//! <summary>Reports the concrete instance size in bytes, excluding separately allocated storage.</summary>
{attribute 'monitoring' := 'call'}
PROPERTY SelfSize : ULINT
GET
SelfSize := XSIZEOF(THIS^);
END_GET
END_PROPERTY

END_FUNCTION_BLOCK

// ---- Tests/Files/FileByteOperationsTest.TcPOU
(*
SPDX-FileCopyrightText: © 2026 Oleksandr Tiutyk <trofimich@gmail.com>
SPDX-License-Identifier: MIT
License: https://opensource.org/license/mit
*)

(*!
<summary>Exercises queued binary I/O and standalone collision, load, rename and delete operations.</summary>
<description>
Uses one exclusive directory and bounded persistent buffers. Checks short read, EOF, tell and guarded results
before and after cancellation. Independent directory probes must preserve the sentinel file. Rename and delete
are followed by readback and a failed load. Direct operations are drained before the base attempts removal.
Use from one task and keep the case alive until cleanup finishes. Do not copy this test.
</description>
*)

{attribute 'no_assign'}
{attribute 'no_explicit_call' := 'do not call this function block directly'}
FUNCTION_BLOCK FileByteOperationsTest EXTENDS FileContentScenarioTest
VAR_STAT
	//! <summary>Class name shared by instances of this concrete function block.</summary>
	{attribute 'hide'}
	_ClassName : STRING := __POUNAME();
END_VAR
VAR CONSTANT
	//! <summary>Truncates the file and permits binary writes and reads through the same handle.</summary>
	_UpdateBinaryMode : DWORD := Tc2_System.Global_Variables.FOPEN_MODEWRITE
		OR Tc2_System.Global_Variables.FOPEN_MODEPLUS
		OR Tc2_System.Global_Variables.FOPEN_MODEBINARY;
	//! <summary>Marks bytes beyond the written range so partial and empty reads can detect stray writes.</summary>
	_UnusedByte : BYTE := BYTE#16#A5;
END_VAR
VAR
	_Phase : FILE_OPERATIONS_TEST_PHASE;
	_ReusedTask : TOF_Tasks.ITask;
	_Write : TOF_FileSystem.WriteBytesToFile(name := "Write four bytes");
	_TellAfterWrite : TOF_FileSystem.GetPositionInFile(name := "Tell after write");
	_Seek : TOF_FileSystem.SetPositionInFile(name := "Rewind binary file");
	_Read : TOF_FileSystem.ReadBytesFromFile(name := "Short binary read");
	_TellAfterRead : TOF_FileSystem.GetPositionInFile(name := "Tell after read");
	_ReadEof : TOF_FileSystem.ReadBytesFromFile(name := "Read past EOF");
	_CheckEof : TOF_FileSystem.CheckEndOfFile(name := "Check EOF");

	_CheckDirectory : TOF_FileSystem.CheckDirectoryExists(name := "Check file as directory");
	_CreateIfAbsent : TOF_FileSystem.CreateDirectoryIfNotExists(name := "Create on file collision");
	_RemoveIfPresent : TOF_FileSystem.RemoveEmptyDirectoryIfExists(name := "Remove on file collision");
	_CreateExisting : TOF_FileSystem.CreateDirectory(name := "Create existing directory");
	_Load : TOF_FileSystem.LoadFile(name := "Load binary file");
	_Rename : TOF_FileSystem.RenameFile(name := "Rename binary file");
	_Delete : TOF_FileSystem.DeleteFile(name := "Delete binary file");

	_ResultTasks : ARRAY [0..5] OF TOF_Tasks.ITask :=
		[_Write, _TellAfterWrite, _Read, _TellAfterRead, _ReadEof, _CheckEof];
	_CollisionTasks : ARRAY [0..3] OF TOF_Tasks.ITask :=
		[_CheckDirectory, _CreateIfAbsent, _RemoveIfPresent, _CreateExisting];

	_Data : ARRAY [0..3] OF BYTE := [BYTE#16#41, BYTE#16#42, BYTE#16#43, BYTE#16#44];
	_ReadBuffer : ARRAY [0..7] OF BYTE;
	_LoadBuffer : ARRAY [0..7] OF BYTE;
	_EofBuffer : BYTE;
END_VAR

(*!
<summary>Rearms the direct and queued tasks and restores the initial binary buffers.</summary>
*)
METHOD PROTECTED ResetScenario : BOOL
VAR
	i : DINT;
END_VAR
_Phase := FILE_OPERATIONS_TEST_PHASE.START_WRITE;
_ReusedTask := 0;
_EofBuffer := _UnusedByte;

FOR i := LOWER_BOUND(_ReadBuffer, 1) TO UPPER_BOUND(_ReadBuffer, 1) DO
	_ReadBuffer[i] := _UnusedByte;
END_FOR

FOR i := LOWER_BOUND(_ResultTasks, 1) TO UPPER_BOUND(_ResultTasks, 1) DO
	IF NOT _ResultTasks[i].Reset() THEN
		RETURN;
	END_IF
END_FOR

FOR i := LOWER_BOUND(_CollisionTasks, 1) TO UPPER_BOUND(_CollisionTasks, 1) DO
	IF NOT _CollisionTasks[i].Reset() THEN
		RETURN;
	END_IF
END_FOR

ResetScenario := _Seek.Reset() AND_THEN _Load.Reset() AND_THEN _Rename.Reset() AND_THEN _Delete.Reset();
END_METHOD

(*!
<summary>Drains direct and pre-submission cancellation tasks before owned directory removal.</summary>
<description>The base invokes this after the manager stops. Every eligible task is advanced on each call.</description>
*)
METHOD PROTECTED DrainScenario : BOOL
VAR
	i : DINT;
END_VAR
DrainScenario := TRUE;

FOR i := LOWER_BOUND(_CollisionTasks, 1) TO UPPER_BOUND(_CollisionTasks, 1) DO
	DrainScenario := drainTask(task := _CollisionTasks[i]) AND DrainScenario;
END_FOR

IF _ReusedTask <> 0 THEN
	DrainScenario := drainTask(task := _ReusedTask) AND DrainScenario;
END_IF

DrainScenario := drainTask(task := _Load) AND DrainScenario;
DrainScenario := drainTask(task := _Rename) AND DrainScenario;
DrainScenario := drainTask(task := _Delete) AND DrainScenario;
END_METHOD

(*!
<summary>Requests cooperative cancellation and advances an active task one cycle.</summary>
<param name="task">Live task that is no longer controlled by the file manager.</param>
*)
METHOD PRIVATE drainTask : BOOL
VAR_INPUT
	task : TOF_Tasks.ITask;
END_VAR
IF task.State.Running THEN
	task.Cancel();
	task.Execute();
END_IF

drainTask := NOT task.State.Running;
END_METHOD

(*!
<summary>Advances the native byte, collision and path-operation phases.</summary>
<description>Returns TRUE after the final missing-file check. The base handles reporting after cleanup.</description>
*)
METHOD PROTECTED AdvanceScenario : BOOL
VAR
	i : DINT;
END_VAR
CASE _Phase OF
	FILE_OPERATIONS_TEST_PHASE.START_WRITE:
		startByteQueue();

	FILE_OPERATIONS_TEST_PHASE.WAIT_FOR_WRITE:
		_Manager.Execute();

		IF _Write.State.Running THEN
			CheckScenario(
				condition := _Write.ActuallyWrittenBytes = TOF_Core.UnsignedInt32.ZERO,
				message := "RUNNING write must hide its byte count"
			);
		END_IF

		IF _Read.State.Running THEN
			CheckScenario(
				condition := _Read.ActuallyReadBytes = TOF_Core.UnsignedInt32.ZERO AND_THEN NOT _Read.IsEndOfFile,
				message := "RUNNING read must hide its byte count and EOF"
			);
		END_IF

		IF _TellAfterWrite.State.Running THEN
			CheckScenario(
				condition := _TellAfterWrite.Position = TOF_Core.SignedInt32.ZERO,
				message := "RUNNING tell must hide its file position"
			);
		END_IF

		IF _Manager.State.Stopped AND_THEN _ScenarioFailure = "" THEN
			IF checkWorkDone(task := _Manager) THEN
				checkByteResults();
			END_IF

			_Phase := FILE_OPERATIONS_TEST_PHASE.CHECK_COLLISIONS;
		END_IF

	FILE_OPERATIONS_TEST_PHASE.CHECK_COLLISIONS:
		startCollisions();

	FILE_OPERATIONS_TEST_PHASE.WAIT_FOR_COLLISIONS:
		IF checkCollisions() THEN
			_Phase := FILE_OPERATIONS_TEST_PHASE.START_LOAD;
		END_IF

	FILE_OPERATIONS_TEST_PHASE.START_LOAD:
		_Load.TargetBuffer := ADR(_LoadBuffer);
		_Load.TargetBufferSize := SIZEOF(_LoadBuffer);
		_Load.Timeout := _NativeTimeout;
		startLoad(filePath := _Directory.FirstFilePath);
		_Phase := FILE_OPERATIONS_TEST_PHASE.WAIT_FOR_LOAD;

	FILE_OPERATIONS_TEST_PHASE.WAIT_FOR_LOAD:
		_Load.Execute();

		IF _Load.State.Running THEN
			CheckScenario(
				condition := _Load.LoadedBytesCount = TOF_Core.UnsignedInt32.ZERO,
				message := "RUNNING load must hide its byte count"
			);
		ELSIF _Load.State.Stopped AND_THEN checkWorkDone(task := _Load) THEN
			checkLoadedBytes(context := "File after collision attempts");
			_Phase := FILE_OPERATIONS_TEST_PHASE.START_RENAME;
		END_IF

	FILE_OPERATIONS_TEST_PHASE.START_RENAME:
		_Directory.ExpectSecondFile();
		_Rename.OldFilePath := _Directory.FirstFilePath;
		_Rename.NewFilePath := _Directory.SecondFilePath;
		_Rename.PathType := Tc2_System.E_OpenPath.PATH_GENERIC;
		_Rename.Timeout := _NativeTimeout;
		CheckScenario(condition := _Rename.Start(), message := "Rename refused Start");
		_Phase := FILE_OPERATIONS_TEST_PHASE.WAIT_FOR_RENAME;

	FILE_OPERATIONS_TEST_PHASE.WAIT_FOR_RENAME:
		_Rename.Execute();

		IF _Rename.State.Stopped AND_THEN checkWorkDone(task := _Rename) THEN
			_Directory.ConfirmFirstFileAbsent();
			_Phase := FILE_OPERATIONS_TEST_PHASE.LOAD_RENAMED_FILE;
		END_IF

	FILE_OPERATIONS_TEST_PHASE.LOAD_RENAMED_FILE:
		startLoad(filePath := _Directory.SecondFilePath);
		_Phase := FILE_OPERATIONS_TEST_PHASE.WAIT_FOR_RENAMED_LOAD;

	FILE_OPERATIONS_TEST_PHASE.WAIT_FOR_RENAMED_LOAD:
		_Load.Execute();

		IF _Load.State.Stopped AND_THEN checkWorkDone(task := _Load) THEN
			checkLoadedBytes(context := "Renamed file");
			_Phase := FILE_OPERATIONS_TEST_PHASE.START_DELETE;
		END_IF

	FILE_OPERATIONS_TEST_PHASE.START_DELETE:
		_Delete.FilePath := _Directory.SecondFilePath;
		_Delete.PathType := Tc2_System.E_OpenPath.PATH_GENERIC;
		_Delete.Timeout := _NativeTimeout;
		CheckScenario(condition := _Delete.Start(), message := "Delete refused Start");
		_Phase := FILE_OPERATIONS_TEST_PHASE.WAIT_FOR_DELETE;

	FILE_OPERATIONS_TEST_PHASE.WAIT_FOR_DELETE:
		_Delete.Execute();

		IF _Delete.State.Stopped AND_THEN checkWorkDone(task := _Delete) THEN
			_Directory.ConfirmSecondFileAbsent();
			_Phase := FILE_OPERATIONS_TEST_PHASE.LOAD_DELETED_FILE;
		END_IF

	FILE_OPERATIONS_TEST_PHASE.LOAD_DELETED_FILE:
		startLoad(filePath := _Directory.SecondFilePath);
		_Phase := FILE_OPERATIONS_TEST_PHASE.WAIT_FOR_MISSING_LOAD;

	FILE_OPERATIONS_TEST_PHASE.WAIT_FOR_MISSING_LOAD:
		_Load.Execute();

		IF _Load.State.Stopped THEN
			CheckScenario(
				condition := _Load.FinalStopReason.Failure
					AND_THEN _Load.LoadedBytesCount = TOF_Core.UnsignedInt32.ZERO,
				message := "Load of a deleted file must fail and expose zero bytes"
			);

			FOR i := LOWER_BOUND(_LoadBuffer, 1) TO UPPER_BOUND(_LoadBuffer, 1) DO
				IF _LoadBuffer[i] <> _UnusedByte THEN
					CheckScenario(
						condition := FALSE,
						message := TOF_Core.WideStrings.ConcatFit255("Missing-file load altered buffer byte ", TO_WSTRING(i))
					);
					RETURN;
				END_IF
			END_FOR

			AdvanceScenario := TRUE;
		END_IF
END_CASE
END_METHOD

(*!
<summary>Configures and starts the binary write, seek, read and position queue.</summary>
<description>The directory is owned and all borrowed queue tasks are READY.</description>
*)
METHOD PRIVATE startByteQueue
_Directory.ExpectFirstFile();
ConfigureFile(filePath := _Directory.FirstFilePath, modeFlags := _UpdateBinaryMode);
_Write.SourceBuffer := ADR(_Data);
_Write.BytesCountToWrite := SIZEOF(_Data);
_Write.Timeout := _NativeTimeout;
_TellAfterWrite.Timeout := _NativeTimeout;
_Seek.Position := TOF_Core.SignedInt32.ZERO;
_Seek.Origin := Tc2_System.E_SeekOrigin.SEEK_SET;
_Seek.Timeout := _NativeTimeout;
_Read.TargetBuffer := ADR(_ReadBuffer);
_Read.BytesCountToRead := SIZEOF(_ReadBuffer);
_Read.Timeout := _NativeTimeout;
_TellAfterRead.Timeout := _NativeTimeout;
_ReadEof.TargetBuffer := ADR(_EofBuffer);
_ReadEof.BytesCountToRead := SIZEOF(_EofBuffer);
_ReadEof.Timeout := _NativeTimeout;
_CheckEof.Timeout := _NativeTimeout;

_Manager.Enqueue(fileHandleTask := _Write);
_Manager.Enqueue(fileHandleTask := _TellAfterWrite);
_Manager.Enqueue(fileHandleTask := _Seek);
_Manager.Enqueue(fileHandleTask := _Read);
_Manager.Enqueue(fileHandleTask := _TellAfterRead);
_Manager.Enqueue(fileHandleTask := _ReadEof);
_Manager.Enqueue(fileHandleTask := _CheckEof);

CheckScenario(
	condition := _Write.ActuallyWrittenBytes = TOF_Core.UnsignedInt32.ZERO,
	message := "READY write must expose zero bytes"
);
CheckScenario(
	condition := _Read.ActuallyReadBytes = TOF_Core.UnsignedInt32.ZERO AND_THEN NOT _Read.IsEndOfFile,
	message := "READY read must expose zero bytes and FALSE EOF"
);
CheckScenario(condition := NOT _CheckEof.IsEndOfFile, message := "READY EOF query must expose FALSE");

IF _ScenarioFailure = "" THEN
	CheckScenario(condition := _Manager.Start(), message := "Binary write/read queue refused Start");
	_Phase := FILE_OPERATIONS_TEST_PHASE.WAIT_FOR_WRITE;
END_IF
END_METHOD

(*!
<summary>Verifies the readback and neutral results after pre-submission cancellation.</summary>
<description>Call after the manager completes the full queue and releases the resource.</description>
*)
METHOD PRIVATE checkByteResults
VAR
	i : DINT;
	task : TOF_Tasks.ITask;
END_VAR
CheckScenario(
	condition := _Write.ActuallyWrittenBytes = 4,
	message := "Full write must report four bytes"
);
CheckScenario(condition := _Read.ActuallyReadBytes = 4, message := "Short read must report the actual four bytes");
CheckScenario(condition := _TellAfterWrite.Position = 4, message := "Tell after write must report position four");
CheckScenario(condition := _TellAfterRead.Position = 4, message := "Tell after short read must report position four");
CheckScenario(
	condition := _ReadEof.ActuallyReadBytes = TOF_Core.UnsignedInt32.ZERO AND_THEN _ReadEof.IsEndOfFile,
	message := "Read past the data must return zero bytes and TRUE EOF"
);
CheckScenario(condition := _CheckEof.IsEndOfFile, message := "EOF query after empty read must report TRUE");
CheckScenario(condition := _EofBuffer = _UnusedByte, message := "Empty read must preserve its destination");

FOR i := LOWER_BOUND(_Data, 1) TO UPPER_BOUND(_Data, 1) DO
	CheckScenario(
		condition := _ReadBuffer[i] = _Data[i],
		message := TOF_Core.WideStrings.ConcatFit255("Binary readback differs at byte ", TO_WSTRING(i))
	);
END_FOR

FOR i := UPPER_BOUND(_Data, 1) + 1 TO UPPER_BOUND(_ReadBuffer, 1) DO
	CheckScenario(
		condition := _ReadBuffer[i] = _UnusedByte,
		message := TOF_Core.WideStrings.ConcatFit255("Short read altered buffer tail at byte ", TO_WSTRING(i))
	);
END_FOR

IF _ScenarioFailure <> "" THEN
	RETURN;
END_IF

FOR i := LOWER_BOUND(_ResultTasks, 1) TO UPPER_BOUND(_ResultTasks, 1) DO
	task := _ResultTasks[i];
	_ReusedTask := task;

	IF NOT task.Reset() OR_ELSE NOT task.Start() OR_ELSE NOT task.Cancel() THEN
		_ScenarioFailure := TOF_Core.WideStrings.ConcatFit255(task.Name, " refused Reset, Start or Cancel during reuse");
		RETURN;
	END_IF

	task.Execute();

	IF NOT task.State.Stopped OR_ELSE NOT task.FinalStopReason.ExternalCancel THEN
		_ScenarioFailure := TOF_Core.WideStrings.ConcatFit255(
			task.Name, " did not stop with pre-submission cancellation"
		);
		RETURN;
	END_IF

	_ReusedTask := 0;
END_FOR

CheckScenario(
	condition := _Write.ActuallyWrittenBytes = TOF_Core.UnsignedInt32.ZERO,
	message := "Cancelled write exposed its previous byte count"
);
CheckScenario(
	condition := _Read.ActuallyReadBytes = TOF_Core.UnsignedInt32.ZERO,
	message := "Cancelled read exposed its previous byte count"
);
CheckScenario(
	condition := _TellAfterWrite.Position = TOF_Core.SignedInt32.ZERO
		AND_THEN _TellAfterRead.Position = TOF_Core.SignedInt32.ZERO,
	message := "Cancelled tell exposed its previous file position"
);
CheckScenario(condition := NOT _ReadEof.IsEndOfFile, message := "Cancelled read exposed its previous TRUE EOF");
CheckScenario(
	condition := NOT _CheckEof.IsEndOfFile,
	message := "Cancelled EOF query exposed its previous TRUE EOF"
);
END_METHOD

(*!
<summary>Starts directory probes against the existing sentinel file and its parent.</summary>
<description>Only the original fixture owns the directory. All four probes borrow paths only.</description>
*)
METHOD PRIVATE startCollisions
VAR
	i : DINT;
END_VAR
_CheckDirectory.DirectoryPath := _Directory.FirstFilePath;
_CreateIfAbsent.DirectoryPath := _Directory.FirstFilePath;
_RemoveIfPresent.DirectoryPath := _Directory.FirstFilePath;
_CreateExisting.DirectoryPath := _Directory.DirectoryPath;
_CheckDirectory.PathType := Tc2_System.E_OpenPath.PATH_GENERIC;
_CreateIfAbsent.PathType := Tc2_System.E_OpenPath.PATH_GENERIC;
_RemoveIfPresent.PathType := Tc2_System.E_OpenPath.PATH_GENERIC;
_CreateExisting.PathType := Tc2_System.E_OpenPath.PATH_GENERIC;
_CheckDirectory.Timeout := _NativeTimeout;
_CreateIfAbsent.Timeout := _NativeTimeout;
_RemoveIfPresent.Timeout := _NativeTimeout;
_CreateExisting.Timeout := _NativeTimeout;

FOR i := LOWER_BOUND(_CollisionTasks, 1) TO UPPER_BOUND(_CollisionTasks, 1) DO
	IF NOT _CollisionTasks[i].Start() THEN
		_ScenarioFailure := TOF_Core.WideStrings.ConcatFit255(_CollisionTasks[i].Name, " refused Start");
		RETURN;
	END_IF
END_FOR

_Phase := FILE_OPERATIONS_TEST_PHASE.WAIT_FOR_COLLISIONS;
END_METHOD

(*!
<summary>Advances outstanding collision probes and verifies their stopped results.</summary>
<description>Returns TRUE after all four operations stop with the expected outcomes.</description>
*)
METHOD PRIVATE checkCollisions : BOOL
VAR
	i : DINT;
	allStopped : BOOL := TRUE;
END_VAR
FOR i := LOWER_BOUND(_CollisionTasks, 1) TO UPPER_BOUND(_CollisionTasks, 1) DO
	IF _CollisionTasks[i].State.Running THEN
		_CollisionTasks[i].Execute();
	END_IF

	allStopped := allStopped AND _CollisionTasks[i].State.Stopped;
END_FOR

IF NOT allStopped THEN
	RETURN;
END_IF

IF NOT checkWorkDone(task := _CheckDirectory) THEN
	RETURN;
END_IF

CheckScenario(condition := NOT _CheckDirectory.DirectoryExists, message := "A file was reported as a directory");
CheckScenario(
	condition := _CreateIfAbsent.FinalStopReason.Failure,
	message := "Conditional directory creation did not reject the file collision"
);
CheckScenario(
	condition := _RemoveIfPresent.FinalStopReason.Failure,
	message := "Conditional directory removal did not reject the file collision"
);
CheckScenario(
	condition := _CreateExisting.FinalStopReason.Failure,
	message := "Ordinary directory creation did not reject the existing directory"
);
checkCollisions := _ScenarioFailure = "";
END_METHOD

(*!
<summary>Resets the load task, refills its target and starts loading the specified file.</summary>
<param name="filePath">Owned fixture path to load, including the deliberate missing-file check.</param>
*)
METHOD PRIVATE startLoad
VAR_INPUT
	filePath : Tc2_System.T_MaxString;
END_VAR
VAR
	i : DINT;
END_VAR
IF NOT _Load.Reset() THEN
	_ScenarioFailure := "File load refused Reset";
	RETURN;
END_IF

IF _Load.LoadedBytesCount <> TOF_Core.UnsignedInt32.ZERO THEN
	_ScenarioFailure := "READY file load exposed its previous byte count";
	RETURN;
END_IF

FOR i := LOWER_BOUND(_LoadBuffer, 1) TO UPPER_BOUND(_LoadBuffer, 1) DO
	_LoadBuffer[i] := _UnusedByte;
END_FOR

_Load.FilePath := filePath;
CheckScenario(condition := _Load.Start(), message := "File load refused Start");
END_METHOD

(*!
<summary>Checks the full sentinel and the untouched tail of a successful load.</summary>
<param name="context">Operation that preceded this readback.</param>
*)
METHOD PRIVATE checkLoadedBytes
VAR_INPUT
	context : WSTRING(80);
END_VAR
VAR
	i : DINT;
END_VAR
CheckScenario(
	condition := _Load.LoadedBytesCount = 4,
	message := TOF_Core.WideStrings.ConcatFit255(context, ": expected four loaded bytes")
);

FOR i := LOWER_BOUND(_Data, 1) TO UPPER_BOUND(_Data, 1) DO
	CheckScenario(
		condition := _LoadBuffer[i] = _Data[i],
		message := TOF_Core.WideStrings.ConcatFit255(context, ": sentinel differs at byte ", TO_WSTRING(i))
	);
END_FOR

FOR i := UPPER_BOUND(_Data, 1) + 1 TO UPPER_BOUND(_LoadBuffer, 1) DO
	CheckScenario(
		condition := _LoadBuffer[i] = _UnusedByte,
		message := TOF_Core.WideStrings.ConcatFit255(context, ": load altered buffer tail at byte ", TO_WSTRING(i))
	);
END_FOR
END_METHOD

(*!
<summary>Reports the task name and copied stop diagnostic when a native operation fails.</summary>
<param name="task">Stopped task whose success is required to continue.</param>
*)
METHOD PRIVATE checkWorkDone : BOOL
VAR_INPUT
	task : TOF_Tasks.ITask;
END_VAR
checkWorkDone := task.FinalStopReason.WorkDone;

IF NOT checkWorkDone AND_THEN _ScenarioFailure = "" THEN
	_ScenarioFailure := TOF_Core.WideStrings.ConcatFit255(task.Name, " did not finish with WorkDone: ");
	TOF_Core.WideStrings.AppendFit(targetString := _ScenarioFailure, sourceString := task.FinalStopReason.Message);
END_IF
END_METHOD

//! <summary>Borrows the concrete type name; callers must not modify the referenced storage.</summary>
{attribute 'monitoring' := 'call'}
PROPERTY ClassName : REFERENCE TO STRING
GET
ClassName REF= _ClassName;
END_GET
END_PROPERTY

//! <summary>Borrows the compiler-initialized namespace; callers must not modify it.</summary>
{attribute 'monitoring' := 'call'}
PROPERTY NamespaceName : REFERENCE TO STRING
GET
NamespaceName REF= CurrentNamespace.Name;
END_GET
END_PROPERTY

//! <summary>Reports the concrete instance size in bytes, excluding separately allocated storage.</summary>
{attribute 'monitoring' := 'call'}
PROPERTY SelfSize : ULINT
GET
SelfSize := XSIZEOF(THIS^);
END_GET
END_PROPERTY

END_FUNCTION_BLOCK

// ---- Tests/Files/FileBinaryBufferMatrixTest.TcPOU
(*
SPDX-FileCopyrightText: © 2026 Oleksandr Tiutyk <trofimich@gmail.com>
SPDX-License-Identifier: MIT
License: https://opensource.org/license/mit
*)

(*!
<summary>Checks six invalid binary buffer configurations on an acquired file resource.</summary>
<description>
Uses an owned file and opens a fresh update handle for each row. Verifies the configured property diagnostic,
neutral public results, intact caller data and resource release. No sampled cycle may report native busy;
native tracing is needed to rule out a submission that completed between observations.
Use from one task and do not copy this test.
</description>
*)

{attribute 'no_assign'}
{attribute 'no_explicit_call' := 'do not call this function block directly'}
FUNCTION_BLOCK FileBinaryBufferMatrixTest EXTENDS FileContentScenarioTest
VAR_STAT
	//! <summary>Class name shared by instances of this concrete function block.</summary>
	{attribute 'hide'}
	_ClassName : STRING := __POUNAME();
END_VAR
VAR CONSTANT
	//! <summary>First row using WriteBytesToFile. The preceding three rows use ReadBytesFromFile.</summary>
	_FirstWriteRow : DINT := 3;
	//! <summary>Total number of null and zero sized buffer configurations under test.</summary>
	_RowCount : DINT := 6;
	//! <summary>Identifies unexpected changes to caller-owned storage in each invalid row.</summary>
	_BufferSentinel : BYTE := BYTE#16#A5;
	//! <summary>Creates a new, empty binary file before the validation rows.</summary>
	_CreateBinaryMode : DWORD := Tc2_System.Global_Variables.FOPEN_MODEWRITE
		OR Tc2_System.Global_Variables.FOPEN_MODEBINARY;
	//! <summary>Reopens the existing file for binary reads and writes without truncating it.</summary>
	_OpenBinaryMode : DWORD := Tc2_System.Global_Variables.FOPEN_MODEREAD
		OR Tc2_System.Global_Variables.FOPEN_MODEPLUS
		OR Tc2_System.Global_Variables.FOPEN_MODEBINARY;
END_VAR
VAR
	_Phase : FILE_BUFFER_TEST_PHASE;
	_Read : TOF_FileSystem.ReadBytesFromFile(name := "Invalid read buffer");
	_Write : TOF_FileSystem.WriteBytesToFile(name := "Invalid write buffer");
	_Operation : TOF_Tasks.ITask;
	_ExpectedProperty : STRING(32);
	_Row : DINT;
	_Buffer : BYTE;
END_VAR

(*!
<summary>Rearms the binary operations and restarts the matrix from its first row.</summary>
*)
METHOD PROTECTED ResetScenario : BOOL
_Phase := FILE_BUFFER_TEST_PHASE.CREATE_FILE;
_Operation := 0;
_Row := 0;
ResetScenario := _Read.Reset() AND_THEN _Write.Reset();
END_METHOD

(*!
<summary>Creates the fixture file and advances one invalid buffer row at a time.</summary>
<description>Queues the invalid child only after acquisition is observed. Returns TRUE after the sixth row.</description>
*)
METHOD PROTECTED AdvanceScenario : BOOL
CASE _Phase OF
	FILE_BUFFER_TEST_PHASE.CREATE_FILE:
		_Directory.ExpectFirstFile();
		ConfigureFile(filePath := _Directory.FirstFilePath, modeFlags := _CreateBinaryMode);
		CheckScenario(condition := _Manager.Start(), message := "Creating the matrix file refused Start");
		_Phase := FILE_BUFFER_TEST_PHASE.WAIT_FOR_FILE;

	FILE_BUFFER_TEST_PHASE.WAIT_FOR_FILE:
		_Manager.Execute();

		IF _Manager.State.Stopped THEN
			IF NOT _Manager.FinalStopReason.WorkDone OR_ELSE _Manager.ResourceManager.ResourceAcquired THEN
				_ScenarioFailure := "Creating the matrix file did not finish and release the resource: ";
				TOF_Core.WideStrings.AppendFit(
					targetString := _ScenarioFailure,
					sourceString := _Manager.FinalStopReason.Message
				);
				RETURN;
			END_IF

			_Phase := FILE_BUFFER_TEST_PHASE.START_INVALID_OPERATION;
		END_IF

	FILE_BUFFER_TEST_PHASE.START_INVALID_OPERATION:
		startRow();

	FILE_BUFFER_TEST_PHASE.WAIT_FOR_INVALID_OPERATION:
		_Manager.Execute();

		IF _Manager.State.Stopped THEN
			IF NOT checkRow() THEN
				RETURN;
			END_IF

			_Row := _Row + 1;
			AdvanceScenario := _Row = _RowCount;
			_Phase := FILE_BUFFER_TEST_PHASE.START_INVALID_OPERATION;
		ELSIF _Read.FileOperationInProgress OR_ELSE _Write.FileOperationInProgress THEN
			failRow(reason := "an invalid buffer exposed a pending native request");
		ELSIF _Manager.ResourceManager.ResourceAcquired
			AND_THEN _Manager.RunningSubstate.Processing
			AND_THEN _Manager.PendingTaskCount = 0
			AND_THEN _Operation.State.Ready
		THEN
			IF _Row < _FirstWriteRow THEN
				_Manager.Enqueue(fileHandleTask := _Read);
			ELSE
				_Manager.Enqueue(fileHandleTask := _Write);
			END_IF

			_Manager.StopWhenNoPendingTasks := TRUE;
		END_IF
END_CASE
END_METHOD

(*!
<summary>Configures one null or zero buffer combination and starts acquiring its file.</summary>
<description>Called with no active file operation, after creating the file or checking the previous row.</description>
*)
METHOD PRIVATE startRow
IF NOT _Manager.Reset() OR_ELSE NOT _Read.Reset() OR_ELSE NOT _Write.Reset() THEN
	_ScenarioFailure := TOF_Core.WideStrings.ConcatFit255(
		"Buffer row ", TO_WSTRING(_Row + 1), ": the manager or a binary operation refused Reset"
	);
	RETURN;
END_IF

ConfigureFile(filePath := _Directory.FirstFilePath, modeFlags := _OpenBinaryMode);
_Manager.StopWhenNoPendingTasks := FALSE;
_Buffer := _BufferSentinel;
_Read.Timeout := _NativeTimeout;
_Write.Timeout := _NativeTimeout;
_Read.TargetBuffer := TOF_Core.Memory.NULL_ADDRESS;
_Read.BytesCountToRead := TOF_Core.UnsignedInt32.ZERO;
_Write.SourceBuffer := TOF_Core.Memory.NULL_ADDRESS;
_Write.BytesCountToWrite := TOF_Core.UnsignedInt32.ZERO;

CASE _Row OF
	0:
		_Read.BytesCountToRead := 1;
		_ExpectedProperty := 'TargetBuffer';
	1:
		_Read.TargetBuffer := ADR(_Buffer);
		_ExpectedProperty := 'BytesCountToRead';
	2:
		_ExpectedProperty := 'TargetBuffer';
	3:
		_Write.BytesCountToWrite := 1;
		_ExpectedProperty := 'SourceBuffer';
	4:
		_Write.SourceBuffer := ADR(_Buffer);
		_ExpectedProperty := 'BytesCountToWrite';
	5:
		_ExpectedProperty := 'SourceBuffer';
END_CASE

IF _Row < _FirstWriteRow THEN
	_Operation := _Read;
ELSE
	_Operation := _Write;
END_IF

IF NOT _Manager.Start() THEN
	failRow(reason := "the update file manager refused Start");
	RETURN;
END_IF

_Phase := FILE_BUFFER_TEST_PHASE.WAIT_FOR_INVALID_OPERATION;
END_METHOD

(*!
<summary>Verifies the actual child failure, release and data after the manager stops.</summary>
<description>Returns TRUE for a failed child with its expected property diagnostic and no retained resource.</description>
*)
METHOD PRIVATE checkRow : BOOL
VAR
	diagnostic : STRING(255);
END_VAR
IF NOT _Operation.State.Stopped OR_ELSE NOT _Operation.FinalStopReason.Failure THEN
	failRow(reason := "the invalid child did not reach STOPPED with Failure");
	TOF_Core.WideStrings.AppendFit(targetString := _ScenarioFailure, sourceString := " | Manager: ");
	TOF_Core.WideStrings.AppendFit(targetString := _ScenarioFailure, sourceString := _Manager.FinalStopReason.Message);
	RETURN;
END_IF

IF NOT _Manager.FinalStopReason.Failure OR_ELSE _Manager.ResourceManager.ResourceAcquired THEN
	failRow(reason := "the manager did not report Failure with the resource released");
	RETURN;
END_IF

IF _Read.FileOperationInProgress OR_ELSE _Write.FileOperationInProgress THEN
	failRow(reason := "native I/O was still pending after the manager stopped");
	RETURN;
END_IF

IF _Buffer <> _BufferSentinel
	OR_ELSE _Read.ActuallyReadBytes <> TOF_Core.UnsignedInt32.ZERO
	OR_ELSE _Write.ActuallyWrittenBytes <> TOF_Core.UnsignedInt32.ZERO
	OR_ELSE _Read.IsEndOfFile
THEN
	failRow(reason := "the invalid operation altered caller data or exposed a non-neutral result");
	RETURN;
END_IF

diagnostic := TO_STRING(_Operation.FinalStopReason.Message);

IF NOT TOF_Core.Strings.Contains(stringToSearchIn := diagnostic, stringToFind := _ExpectedProperty) THEN
	failRow(reason := "the child diagnostic did not name the expected public property");
	TOF_Core.WideStrings.AppendFit(targetString := _ScenarioFailure, sourceString := " | Actual: ");
	TOF_Core.WideStrings.AppendFit(targetString := _ScenarioFailure, sourceString := _Operation.FinalStopReason.Message);
	RETURN;
END_IF

checkRow := TRUE;
END_METHOD

(*!
<summary>Copies the matrix row, expected property and its first failure for deferred reporting.</summary>
<param name="reason">Condition that failed before cooperative cleanup.</param>
*)
METHOD PRIVATE failRow
VAR_INPUT
	reason : WSTRING(255);
END_VAR
_ScenarioFailure := TOF_Core.WideStrings.ConcatFit255(
	"Buffer row ", TO_WSTRING(_Row + 1), " (", TO_WSTRING(_ExpectedProperty), "): ", reason
);
END_METHOD

//! <summary>Borrows the concrete type name; callers must not modify the referenced storage.</summary>
{attribute 'monitoring' := 'call'}
PROPERTY ClassName : REFERENCE TO STRING
GET
ClassName REF= _ClassName;
END_GET
END_PROPERTY

//! <summary>Borrows the compiler-initialized namespace; callers must not modify it.</summary>
{attribute 'monitoring' := 'call'}
PROPERTY NamespaceName : REFERENCE TO STRING
GET
NamespaceName REF= CurrentNamespace.Name;
END_GET
END_PROPERTY

//! <summary>Reports the concrete instance size in bytes, excluding separately allocated storage.</summary>
{attribute 'monitoring' := 'call'}
PROPERTY SelfSize : ULINT
GET
SelfSize := XSIZEOF(THIS^);
END_GET
END_PROPERTY

END_FUNCTION_BLOCK

// ---- Tests/Files/FileCallerExceptionCleanupTest.TcPOU
(*
SPDX-FileCopyrightText: © 2026 Oleksandr Tiutyk <trofimich@gmail.com>
SPDX-License-Identifier: MIT
License: https://opensource.org/license/mit
*)

(*!
<summary>Verifies cooperative release after an exception in the file manager's caller.</summary>
<description>
Raises a known StandardException only while the file resource is acquired. The caller catches and checks its
identity, then requests cancellation on a later cycle and drives the manager to STOPPED. The base removes the
owned artifacts before publishing a result. Native resource state does not certify physical close.
Use from one task and do not copy this test.
</description>
*)

{attribute 'no_assign'}
{attribute 'no_explicit_call' := 'do not call this function block directly'}
FUNCTION_BLOCK FileCallerExceptionCleanupTest EXTENDS FileContentScenarioTest
VAR_STAT
	//! <summary>Class name shared by instances of this concrete function block.</summary>
	{attribute 'hide'}
	_ClassName : STRING := __POUNAME();
END_VAR
VAR CONSTANT
	//! <summary>Payload used to distinguish the deliberate caller fault from unrelated exceptions.</summary>
	_CallerMessage : WSTRING(255) := "Synthetic exception in the file-scenario caller";
	//! <summary>Creates an empty owned file for observing acquisition and cancellation.</summary>
	_CreateBinaryMode : DWORD := Tc2_System.Global_Variables.FOPEN_MODEWRITE
		OR Tc2_System.Global_Variables.FOPEN_MODEBINARY;
END_VAR
VAR
	_Phase : FILE_CALLER_CLEANUP_TEST_PHASE;
END_VAR

(*!
<summary>Restores the opening phase after the base rearms the manager.</summary>
*)
METHOD PROTECTED ResetScenario : BOOL
_Phase := FILE_CALLER_CLEANUP_TEST_PHASE.OPEN_FILE;
ResetScenario := TRUE;
END_METHOD

(*!
<summary>Opens a file, catches the caller fault and continues cancellation until release.</summary>
<description>Returns TRUE after observing STOPPED and checking the final reason and resource state.</description>
*)
METHOD PROTECTED AdvanceScenario : BOOL
CASE _Phase OF
	FILE_CALLER_CLEANUP_TEST_PHASE.OPEN_FILE:
		_Directory.ExpectFirstFile();
		ConfigureFile(filePath := _Directory.FirstFilePath, modeFlags := _CreateBinaryMode);
		_Manager.StopWhenNoPendingTasks := FALSE;
		CheckScenario(condition := _Manager.Start(), message := "Caller-exception manager refused Start");
		_Phase := FILE_CALLER_CLEANUP_TEST_PHASE.INJECT_CALLER_EXCEPTION;

	FILE_CALLER_CLEANUP_TEST_PHASE.INJECT_CALLER_EXCEPTION:
		_Manager.Execute();

		IF _Manager.State.Running
			AND_THEN _Manager.ResourceManager.ResourceAcquired
			AND_THEN _Manager.RunningSubstate.Processing
		THEN
			CheckScenario(
				condition := catchCallerException(),
				message := "Expected caller exception was not caught intact"
			);
			_Phase := FILE_CALLER_CLEANUP_TEST_PHASE.DRAIN_MANAGER;
		ELSIF _Manager.State.Stopped THEN
			_ScenarioFailure := "Caller fault requires an acquired file resource: ";
			TOF_Core.WideStrings.AppendFit(
				targetString := _ScenarioFailure,
				sourceString := _Manager.FinalStopReason.Message
			);
		END_IF

	FILE_CALLER_CLEANUP_TEST_PHASE.DRAIN_MANAGER:
		IF _Manager.RunningSubstate.Processing AND_THEN NOT _Manager.Cancel() THEN
			_ScenarioFailure := "The acquired manager refused caller cancellation";
			RETURN;
		END_IF

		_Manager.Execute();

		IF _Manager.State.Stopped THEN
			IF NOT _Manager.FinalStopReason.ExternalCancel THEN
				_ScenarioFailure := "Caller recovery did not stop with ExternalCancel: ";
				TOF_Core.WideStrings.AppendFit(
					targetString := _ScenarioFailure,
					sourceString := _Manager.FinalStopReason.Message
				);
				RETURN;
			END_IF

			CheckScenario(
				condition := NOT _Manager.ResourceManager.ResourceAcquired,
				message := "Caller recovery left the file resource acquired"
			);
			AdvanceScenario := TRUE;
		END_IF
END_CASE
END_METHOD

(*!
<summary>Injects and recognises the deliberate exception outside the manager's Execute call.</summary>
<description>Returns TRUE only for the expected standard payload. No exception reference survives this call.</description>
*)
METHOD PRIVATE catchCallerException : BOOL
VAR
	exceptionCode : __SYSTEM.ExceptionCode;
	caughtException : TOF_Core.IException;
	standardException : TOF_Core.IStandardException;
	message : TOF_Core.ERROR_MESSAGE;
END_VAR
message := _CallerMessage;

__TRY
	TOF_Core.Exceptions.ThrowStandard(
		sourceNamespaceName := NamespaceName,
		sourceClassName := ClassName,
		sourcePOUName := __POUNAME(),
		sourcePosition := __POSITION(),
		message := message
	);
__CATCH(exceptionCode)
	caughtException := TOF_Core.ExceptionManager.GetLastException(
		exceptionCode := exceptionCode,
		catchPointNamespaceName := NamespaceName,
		catchPointPOUName := __POUNAME(),
		catchPointPosition := __POSITION()
	);
	catchCallerException := __QUERYINTERFACE(caughtException, standardException)
		AND_THEN standardException.SourceMessage = _CallerMessage;
__ENDTRY
END_METHOD

//! <summary>Borrows the concrete type name; callers must not modify the referenced storage.</summary>
{attribute 'monitoring' := 'call'}
PROPERTY ClassName : REFERENCE TO STRING
GET
ClassName REF= _ClassName;
END_GET
END_PROPERTY

//! <summary>Borrows the compiler-initialized namespace; callers must not modify it.</summary>
{attribute 'monitoring' := 'call'}
PROPERTY NamespaceName : REFERENCE TO STRING
GET
NamespaceName REF= CurrentNamespace.Name;
END_GET
END_PROPERTY

//! <summary>Reports the concrete instance size in bytes, excluding separately allocated storage.</summary>
{attribute 'monitoring' := 'call'}
PROPERTY SelfSize : ULINT
GET
SelfSize := XSIZEOF(THIS^);
END_GET
END_PROPERTY

END_FUNCTION_BLOCK

// ---- Tests/Loggers/LoggerContractTestGroup.TcPOU
(*
SPDX-FileCopyrightText: c 2026 Oleksandr Tiutyk <trofimich@gmail.com>
SPDX-License-Identifier: MIT
License: https://opensource.org/license/mit
*)

(*!
<summary>Groups the deterministic logger contracts and task-routing cases.</summary>
<description>
Owns nine children in a fixed array for single-task use. Children borrows that array. The group must not be
copied.
</description>
*)

{attribute 'no_assign'}
{attribute 'no_explicit_call' := 'do not call this function block directly'}
FUNCTION_BLOCK LoggerContractTestGroup EXTENDS TOF_Testing.TestGroup<9>
VAR_STAT
	{attribute 'hide'}
	_ClassName : STRING := __POUNAME();
END_VAR
VAR
	_QueuedSnapshotsAndFifo : QueuedLoggerSnapshotTest(name := "QueuedSnapshotsAndFifo", parent := THIS^);
	_QueuedCapacityAndWraparound : QueuedLoggerCapacityTest(name := "QueuedCapacityAndWraparound", parent := THIS^);
	_QueuedDeliveryFailures : QueuedLoggerDeliveryFailureTest(name := "QueuedDeliveryFailures", parent := THIS^);
	_FormatterFailureContainment : LoggerFormatterFailureTest(name := "FormatterFailureContainment", parent := THIS^);
	_MetadataAndZeroRecordLimit : LoggerMetadataAndRecordLimitTest(name := "MetadataAndZeroRecordLimit", parent := THIS^);
	_IndependentTaskDiagnostics : LoggerTaskDiagnosticsTest(name := "IndependentTaskDiagnostics", parent := THIS^);
	_AggregateSnapshotsAndPartialAdmission : QueuedLoggerAggregateTest(
		name := "AggregateSnapshotsAndPartialAdmission",
		parent := THIS^
	);
	_CurrentTaskLoggerRouting : CurrentTaskLoggerRoutingTest(name := "CurrentTaskLoggerRouting", parent := THIS^);
	_RejectNonCyclicInitialization : LoggerNonCyclicInitializationTest(
		name := "RejectNonCyclicInitialization",
		parent := THIS^
	);

	_Children : ARRAY [0.._ChildCount - 1] OF TOF_Testing.ITestElement :=
	[
		_QueuedSnapshotsAndFifo,
		_QueuedCapacityAndWraparound,
		_QueuedDeliveryFailures,
		_FormatterFailureContainment,
		_MetadataAndZeroRecordLimit,
		_IndependentTaskDiagnostics,
		_AggregateSnapshotsAndPartialAdmission,
		_CurrentTaskLoggerRouting,
		_RejectNonCyclicInitialization
	];
END_VAR

//! <summary>Borrows the fixed child array. Callers must not modify it.</summary>
{attribute 'monitoring' := 'call'}
PROPERTY Children : REFERENCE TO ARRAY [0.._ChildCount - 1] OF TOF_Testing.ITestElement
GET
Children REF= _Children;
END_GET
END_PROPERTY

//! <summary>Borrows the concrete class name for the instance lifetime. Callers must not modify it.</summary>
{attribute 'monitoring' := 'call'}
PROPERTY ClassName : REFERENCE TO STRING
GET
ClassName REF= _ClassName;
END_GET
END_PROPERTY

//! <summary>Borrows the compiler-initialized namespace. Callers must not modify it.</summary>
{attribute 'monitoring' := 'call'}
PROPERTY NamespaceName : REFERENCE TO STRING
GET
NamespaceName REF= CurrentNamespace.Name;
END_GET
END_PROPERTY

//! <summary>Reports the complete instance size in bytes, excluding separately allocated storage.</summary>
{attribute 'monitoring' := 'call'}
PROPERTY SelfSize : ULINT
GET
SelfSize := XSIZEOF(THIS^);
END_GET
END_PROPERTY

END_FUNCTION_BLOCK

// ---- Tests/Loggers/QueuedLoggerSnapshotTest.TcPOU
(*
SPDX-FileCopyrightText: c 2026 Oleksandr Tiutyk <trofimich@gmail.com>
SPDX-License-Identifier: MIT
License: https://opensource.org/license/mit
*)

(*!
<summary>Checks FIFO delivery and copied message, number and error snapshots.</summary>
<description>
The runner task owns the fixtures. Each run clears its observations and uses the same instances.
</description>
*)

{attribute 'no_assign'}
{attribute 'no_explicit_call' := 'do not call this function block directly'}
FUNCTION_BLOCK QueuedLoggerSnapshotTest EXTENDS TOF_Testing.SingleCycleTest
VAR_STAT
	{attribute 'hide'}
	_ClassName : STRING := __POUNAME();
END_VAR
VAR
	_Queue : TOF_Loggers.QueuedLogger;
	_Backend : LoggerCaptureBackend;
	_QueueConfigured : BOOL;
END_VAR

(*!
<summary>Checks FIFO delivery and copied message, number and error snapshots.</summary>
<description>
The runner task owns the fixtures. Each run clears its observations and uses the same instances.
</description>
*)
METHOD PROTECTED ExecuteTest
VAR
	message : TOF_Core.ERROR_MESSAGE := "first snapshot";
	number : ULINT := 17;
	error : TOF_Core.ERROR;
	expectedError : TOF_Core.ERROR_MESSAGE;
	record : LOGGER_CAPTURED_MESSAGE;
END_VAR
IF NOT _QueueConfigured THEN
	Assert.ThatBool(actual := _Queue.Configure(backend := 0), message := "Queue must reject a null backend").IsFalse();
	Assert.ThatBool(actual := _Queue.Configure(backend := _Queue), message := "Queue must reject itself").IsFalse();
	_QueueConfigured := _Queue.Configure(backend := _Backend);
END_IF

Assert.ThatBool(actual := _QueueConfigured, message := "Queue must bind to its capture backend").IsTrue();

IF NOT _QueueConfigured THEN
	RETURN;
END_IF

Assert.ThatBool(
	actual := _Queue.PendingMessageCount = 0,
	message := "Scenario must start with an empty queue"
).IsTrue();
Assert.ThatBool(
	actual := _Queue.Configure(backend := _Backend),
	message := "Queue must refuse to replace a configured backend"
).IsFalse();

Assert.ThatBool(
	actual := _Queue.TryLogMessage(
		category := TOF_Core.LOG_CATEGORY.WARNING,
		message := message,
		messageNumber := number
	),
	message := "Numbered message must be queued"
).IsTrue();
message := "second snapshot";
number := 29;
Assert.ThatBool(
	actual := _Queue.TryLogMessage(category := TOF_Core.LOG_CATEGORY.DEBUG, message := message),
	message := "Unnumbered message must be queued"
).IsTrue();
error.SetMessage(message := "copied critical error");
error.SetSeverity(severity := TOF_Core.ERROR_SEVERITY.CRITICAL);
expectedError := error.ToString(
	sourceDisplayMode := TOF_Core.ERROR_SOURCE_DISPLAY_MODE.TOP_AND_ROOT,
	timestampDisplayMode := TOF_Core.TIMESTAMP_DISPLAY_MODE.LOCAL
);
Assert.ThatBool(
	actual := _Queue.TryLogError(error := error, messageNumber := number),
	message := "Error must be queued"
).IsTrue();
message := "mutated caller storage";
number := 99;
error.Clear();
Assert.ThatDInt(actual := _Queue.PendingMessageCount, message := "All three snapshots must be pending").ToBe(
	expected := 3
);
Assert.ThatUInt(actual := _Backend.CapturedCount, message := "Admission must not deliver immediately").ToBe(expected := 0);
_Queue.Execute();
Assert.ThatBool(actual := _Backend.CapturedCount = 3, message := "All three records must reach the backend").IsTrue();
record := _Backend.RecordAt(index := 0);
Assert.ThatBool(
	actual := record.Message = "first snapshot",
	message := "First text must survive caller mutation"
).IsTrue();
Assert.ThatBool(
	actual := record.HasMessageNumber AND_THEN record.MessageNumber = 17,
	message := "Number must be copied"
).IsTrue();
Assert.ThatBool(
	actual := record.Category = TOF_Core.LOG_CATEGORY.WARNING,
	message := "First category must be preserved"
).IsTrue();
record := _Backend.RecordAt(index := 1);
Assert.ThatBool(
	actual := record.Message = "second snapshot",
	message := "FIFO order must preserve the second record"
).IsTrue();
Assert.ThatBool(
	actual := record.HasMessageNumber,
	message := "An absent number must not inherit the prior slot number"
).IsFalse();
Assert.ThatBool(
	actual := record.Category = TOF_Core.LOG_CATEGORY.DEBUG,
	message := "Second category must be preserved"
).IsTrue();

record := _Backend.RecordAt(index := 2);
Assert.ThatBool(actual := record.Message = expectedError, message := "Error text must be copied before Clear").IsTrue();
Assert.ThatBool(
	actual := record.Category = TOF_Core.LOG_CATEGORY.CRITICAL_ERROR,
	message := "Critical severity must survive"
).IsTrue();
Assert.ThatBool(
	actual := record.HasMessageNumber AND_THEN record.MessageNumber = 29,
	message := "Error number must be copied"
).IsTrue();
Assert.ThatBool(actual := _Queue.PendingMessageCount = 0, message := "Queue must be empty after delivery").IsTrue();
Assert.ThatBool(
	actual := _Queue.FailedDeliveryCount = 0,
	message := "Successful delivery must not increase failures"
).IsTrue();
END_METHOD

(*!
<summary>Clears capture observations and injected faults before each run.</summary>
*)
METHOD PROTECTED BeforeTest
_Backend.ResetCapture();
END_METHOD

//! <summary>Borrows the concrete class name for the instance lifetime. Callers must not modify it.</summary>
{attribute 'monitoring' := 'call'}
PROPERTY ClassName : REFERENCE TO STRING
GET
ClassName REF= _ClassName;
END_GET
END_PROPERTY

//! <summary>Borrows the compiler-initialized namespace. Callers must not modify it.</summary>
{attribute 'monitoring' := 'call'}
PROPERTY NamespaceName : REFERENCE TO STRING
GET
NamespaceName REF= CurrentNamespace.Name;
END_GET
END_PROPERTY

//! <summary>Reports the complete instance size in bytes, excluding separately allocated storage.</summary>
{attribute 'monitoring' := 'call'}
PROPERTY SelfSize : ULINT
GET
SelfSize := XSIZEOF(THIS^);
END_GET
END_PROPERTY

END_FUNCTION_BLOCK

// ---- Tests/Loggers/LoggerCaptureBackend.TcPOU
(*
SPDX-FileCopyrightText: © 2026 Oleksandr Tiutyk <trofimich@gmail.com>
SPDX-License-Identifier: MIT
License: https://opensource.org/license/mit
*)
(*!
<summary>Captures backend calls and injects explicitly selected delivery faults.</summary>
<description>
One test task owns this fixture and its copied records. THROW_EXCEPTION deliberately violates the ILogger
Try contract to verify that a wrapper contains a hostile backend. Manager regressions temporarily install the
fixture as the current task logger and restore the previous destination before returning. Execute faults are
also intentional; no terminal OOM or lifecycle exception is injected. ResetCapture clears observations and fault
injection between runs.
</description>
*)

{attribute 'no_explicit_call' := 'do not call this function block directly'}
{attribute 'no_assign'}
FUNCTION_BLOCK LoggerCaptureBackend EXTENDS TOF_Core.Object IMPLEMENTS TOF_Core.ILogger
VAR_STAT
	//! <summary>Initialized concrete fixture metadata.</summary>
	_ClassName : STRING := __POUNAME();
END_VAR
VAR CONSTANT
	//! <summary>Captured record slots, sufficient for one default-capacity batch and its regression probes.</summary>
	_CaptureCapacity : UINT := 256;
END_VAR
VAR
	_Records : ARRAY [0.._CaptureCapacity - 1] OF LOGGER_CAPTURED_MESSAGE;
	_CapturedCount : UINT;
	_AttemptCount : UINT;
	_ExecuteCount : UINT;
	_DeliveryBehavior : LOGGER_DELIVERY_BEHAVIOR;
	_ThrowOnExecute : BOOL;
END_VAR

(*!
<summary>Provides the capture fixture AttemptCount observation or setting.</summary>
<description>
Read or configure only from the test owner task between fixture calls.
</description>
*)
PROPERTY AttemptCount : UINT
GET
AttemptCount := _AttemptCount;
END_GET
END_PROPERTY

(*!
<summary>Provides the capture fixture CapturedCount observation or setting.</summary>
<description>
Read or configure only from the test owner task between fixture calls.
</description>
*)
PROPERTY CapturedCount : UINT
GET
CapturedCount := _CapturedCount;
END_GET
END_PROPERTY

(*!
<summary>Borrows the concrete fixture type name.</summary>
<description>
Returns initialized static metadata; do not modify the referenced string.
</description>
*)
{attribute 'monitoring' := 'call'}
PROPERTY ClassName : REFERENCE TO STRING
GET
ClassName REF= _ClassName;
END_GET
END_PROPERTY

(*!
<summary>Provides the capture fixture DeliveryBehavior observation or setting.</summary>
<description>
Read or configure only from the test owner task between fixture calls.
</description>
*)
PROPERTY DeliveryBehavior : LOGGER_DELIVERY_BEHAVIOR
GET
DeliveryBehavior := _DeliveryBehavior;
END_GET
SET
_DeliveryBehavior := DeliveryBehavior;
END_SET
END_PROPERTY

(*!
<summary>Counts service calls and raises only the explicitly requested execution fault.</summary>
*)
METHOD Execute
_ExecuteCount := _ExecuteCount + 1;

IF _ThrowOnExecute THEN
	TOF_Core.Exceptions.ThrowStandard(
		sourceNamespaceName := NamespaceName,
		sourceClassName := ClassName,
		sourcePOUName := __POUNAME(),
		sourcePosition := __POSITION(),
		message := "Injected backend Execute failure"
	);
END_IF
END_METHOD

(*!
<summary>Provides the capture fixture ExecuteCount observation or setting.</summary>
<description>
Read or configure only from the test owner task between fixture calls.
</description>
*)
PROPERTY ExecuteCount : UINT
GET
ExecuteCount := _ExecuteCount;
END_GET
END_PROPERTY

(*!
<summary>Borrows the test namespace.</summary>
<description>
Returns compiler-initialized library storage without ownership transfer.
</description>
*)
{attribute 'monitoring' := 'call'}
PROPERTY NamespaceName : REFERENCE TO STRING
GET
NamespaceName REF= CurrentNamespace.Name;
END_GET
END_PROPERTY

(*!
<summary>Returns a copied capture record at a valid zero-based index.</summary>
<description>
An out-of-range index returns the initialized empty record; no borrowed fixture storage is exposed.
</description>
*)
METHOD RecordAt : LOGGER_CAPTURED_MESSAGE
VAR_INPUT
	index : UINT;
END_VAR
IF index < _CapturedCount THEN
	RecordAt := _Records[index];
END_IF
END_METHOD

(*!
<summary>Reports the concrete fixture size in bytes.</summary>
*)
{attribute 'monitoring' := 'call'}
PROPERTY SelfSize : ULINT
GET
SelfSize := XSIZEOF(THIS^);
END_GET
END_PROPERTY

(*!
<summary>Provides the capture fixture ThrowOnExecute observation or setting.</summary>
<description>
Read or configure only from the test owner task between fixture calls.
</description>
*)
PROPERTY ThrowOnExecute : BOOL
GET
ThrowOnExecute := _ThrowOnExecute;
END_GET
SET
_ThrowOnExecute := ThrowOnExecute;
END_SET
END_PROPERTY

(*!
<summary>Rejects a diagnostic entry that the text-only wrapper must format before delivery.</summary>
<description>
The regression expects QueuedLogger to call TryLogMessage exclusively.
</description>
*)
METHOD TryLogError : BOOL
VAR_INPUT
	error : REFERENCE TO TOF_Core.ERROR;
	messageNumber : REFERENCE TO ULINT := 0;
END_VAR
TryLogError := FALSE;
END_METHOD

(*!
<summary>Rejects a diagnostic entry that the text-only wrapper must format before delivery.</summary>
<description>
The regression expects QueuedLogger to call TryLogMessage exclusively.
</description>
*)
METHOD TryLogException : BOOL
VAR_INPUT
	exception : TOF_Core.IReadOnlyException;
	severity : TOF_Core.ERROR_SEVERITY;
	messageNumber : REFERENCE TO ULINT := 0;
END_VAR
TryLogException := FALSE;
END_METHOD

(*!
<summary>Captures a delivery attempt, returns the configured outcome or injects a hostile backend exception.</summary>
<description>
The THROW_EXCEPTION branch is intentionally outside a CATCH to exercise the consumer no-throw boundary.
A successful capture owns text and number snapshots; admission failure does not write a capture record.
</description>
*)
METHOD TryLogMessage : BOOL
VAR_INPUT
	category : TOF_Core.LOG_CATEGORY;
END_VAR
VAR_IN_OUT CONSTANT
	message : TOF_Core.ERROR_MESSAGE;
END_VAR
VAR_INPUT
	messageNumber : REFERENCE TO ULINT := 0;
END_VAR
_AttemptCount := _AttemptCount + 1;

CASE _DeliveryBehavior OF
	LOGGER_DELIVERY_BEHAVIOR.REFUSE:
		RETURN;

	LOGGER_DELIVERY_BEHAVIOR.THROW_EXCEPTION:
		TOF_Core.Exceptions.ThrowStandard(
			sourceNamespaceName := NamespaceName,
			sourceClassName := ClassName,
			sourcePOUName := __POUNAME(),
			sourcePosition := __POSITION(),
			message := "Injected backend delivery failure"
		);
END_CASE

IF _CapturedCount >= _CaptureCapacity THEN
	RETURN;
END_IF

_Records[_CapturedCount].Category := category;
_Records[_CapturedCount].Message := message;
_Records[_CapturedCount].HasMessageNumber := __ISVALIDREF(messageNumber);

IF _Records[_CapturedCount].HasMessageNumber THEN
	_Records[_CapturedCount].MessageNumber := messageNumber;
END_IF

_CapturedCount := _CapturedCount + 1;
TryLogMessage := TRUE;
END_METHOD

(*!
<summary>Starts a fresh capture and clears any injected delivery or execution fault.</summary>
<description>
Call from the owning test task between scenarios. Existing slots become inaccessible until overwritten.
This resets only the observer; the queue retains its configuration, storage and delivery counters.
</description>
*)
METHOD ResetCapture
_CapturedCount := 0;
_AttemptCount := 0;
_ExecuteCount := 0;
_DeliveryBehavior := LOGGER_DELIVERY_BEHAVIOR.ACCEPT;
_ThrowOnExecute := FALSE;
END_METHOD

END_FUNCTION_BLOCK

// ---- Tests/Loggers/QueuedLoggerCapacityTest.TcPOU
(*
SPDX-FileCopyrightText: c 2026 Oleksandr Tiutyk <trofimich@gmail.com>
SPDX-License-Identifier: MIT
License: https://opensource.org/license/mit
*)

(*!
<summary>Checks queue capacity, overflow preservation and reuse of the ring buffer.</summary>
<description>
The runner task owns the fixtures. Each run clears its observations and uses the same instances.
</description>
*)

{attribute 'no_assign'}
{attribute 'no_explicit_call' := 'do not call this function block directly'}
FUNCTION_BLOCK QueuedLoggerCapacityTest EXTENDS TOF_Testing.SingleCycleTest
VAR_STAT
	{attribute 'hide'}
	_ClassName : STRING := __POUNAME();
END_VAR
VAR
	_Queue : TOF_Loggers.QueuedLogger;
	_Backend : LoggerCaptureBackend;
	_QueueConfigured : BOOL;
END_VAR

(*!
<summary>Checks queue capacity, overflow preservation and reuse of the ring buffer.</summary>
<description>
The runner task owns the fixtures. Each run clears its observations and uses the same instances.
</description>
*)
METHOD PROTECTED ExecuteTest
VAR
	message : TOF_Core.ERROR_MESSAGE;
	entryLabel : WSTRING(255);
	number : ULINT;
	record : LOGGER_CAPTURED_MESSAGE;
	i : DINT;
	failuresBefore : ULINT;
END_VAR
IF NOT _QueueConfigured THEN
	_QueueConfigured := _Queue.Configure(backend := _Backend);
END_IF

Assert.ThatBool(actual := _QueueConfigured, message := "Queue must bind to its capture backend").IsTrue();

IF NOT _QueueConfigured THEN
	RETURN;
END_IF

Assert.ThatBool(
	actual := _Queue.PendingMessageCount = 0,
	message := "Scenario must start with an empty queue"
).IsTrue();

failuresBefore := _Queue.FailedDeliveryCount;

FOR i := 1 TO TOF_Loggers.Parameters.QUEUED_LOGGER_CAPACITY DO
	number := TO_ULINT(i);
	message := TOF_Core.WideStrings.Concat255("entry ", TO_WSTRING(i));
	Assert.ThatBool(
		actual := _Queue.TryLogMessage(
			category := TOF_Core.LOG_CATEGORY.INFORMATION,
			message := message,
			messageNumber := number
		),
		message := TOF_Core.WideStrings.Concat255("Queue must accept record ", TO_WSTRING(i))
	).IsTrue();
END_FOR

Assert.ThatBool(
	actual := _Queue.TryLogMessage(category := TOF_Core.LOG_CATEGORY.ERROR, message := message),
	message := "Full queue must refuse the next record"
).IsFalse();
_Queue.Execute();
Assert.ThatBool(
	actual := _Backend.AttemptCount = TOF_Loggers.Parameters.QUEUED_LOGGER_CAPACITY,
	message := "Delivery attempts must equal accepted capacity without retrying the overflow"
).IsTrue();

FOR i := 0 TO TO_DINT(TOF_Loggers.Parameters.QUEUED_LOGGER_CAPACITY) - 1 DO
	record := _Backend.RecordAt(index := TO_UINT(i));
	message := TOF_Core.WideStrings.Concat255("entry ", TO_WSTRING(i + 1));
	entryLabel := TOF_Core.WideStrings.Concat255("Full ring record ", TO_WSTRING(i + 1), " must preserve FIFO text");
	Assert.ThatBool(actual := record.Message = message, message := entryLabel).IsTrue();

	entryLabel := TOF_Core.WideStrings.Concat255("Full ring record ", TO_WSTRING(i + 1), " must have its number");
	Assert.ThatBool(
		actual := record.HasMessageNumber AND_THEN record.MessageNumber = TO_ULINT(i + 1),
		message := entryLabel
	).IsTrue();
END_FOR

IF TOF_Loggers.Parameters.QUEUED_LOGGER_CAPACITY > 0 THEN
	message := "after wraparound";
	Assert.ThatBool(
		actual := _Queue.TryLogMessage(category := TOF_Core.LOG_CATEGORY.WARNING, message := message),
		message := "A drained ring must accept a reused slot"
	).IsTrue();
	_Queue.Execute();
	record := _Backend.RecordAt(index := TOF_Loggers.Parameters.QUEUED_LOGGER_CAPACITY);
	Assert.ThatBool(actual := record.Message = message, message := "Reused slot must deliver its new text").IsTrue();
	Assert.ThatBool(actual := record.HasMessageNumber, message := "Reused slot must clear number presence").IsFalse();
END_IF

Assert.ThatBool(actual := _Queue.PendingMessageCount = 0, message := "Refilled queue must drain").IsTrue();
Assert.ThatULInt(actual := _Queue.FailedDeliveryCount, message := "Overflow is an admission refusal").ToBe(
	expected := failuresBefore
);
END_METHOD

(*!
<summary>Clears capture observations and injected faults before each run.</summary>
*)
METHOD PROTECTED BeforeTest
_Backend.ResetCapture();
END_METHOD

//! <summary>Borrows the concrete class name for the instance lifetime. Callers must not modify it.</summary>
{attribute 'monitoring' := 'call'}
PROPERTY ClassName : REFERENCE TO STRING
GET
ClassName REF= _ClassName;
END_GET
END_PROPERTY

//! <summary>Borrows the compiler-initialized namespace. Callers must not modify it.</summary>
{attribute 'monitoring' := 'call'}
PROPERTY NamespaceName : REFERENCE TO STRING
GET
NamespaceName REF= CurrentNamespace.Name;
END_GET
END_PROPERTY

//! <summary>Reports the complete instance size in bytes, excluding separately allocated storage.</summary>
{attribute 'monitoring' := 'call'}
PROPERTY SelfSize : ULINT
GET
SelfSize := XSIZEOF(THIS^);
END_GET
END_PROPERTY

END_FUNCTION_BLOCK

// ---- Tests/Loggers/QueuedLoggerDeliveryFailureTest.TcPOU
(*
SPDX-FileCopyrightText: c 2026 Oleksandr Tiutyk <trofimich@gmail.com>
SPDX-License-Identifier: MIT
License: https://opensource.org/license/mit
*)

(*!
<summary>Checks single-attempt delivery, failure accounting and continued backend service.</summary>
<description>
The runner task owns the fixtures. Each run clears its observations and uses the same instances.
</description>
*)

{attribute 'no_assign'}
{attribute 'no_explicit_call' := 'do not call this function block directly'}
FUNCTION_BLOCK QueuedLoggerDeliveryFailureTest EXTENDS TOF_Testing.SingleCycleTest
VAR_STAT
	{attribute 'hide'}
	_ClassName : STRING := __POUNAME();
END_VAR
VAR
	_Queue : TOF_Loggers.QueuedLogger;
	_Backend : LoggerCaptureBackend;
	_QueueConfigured : BOOL;
END_VAR

(*!
<summary>Checks single-attempt delivery, failure accounting and continued backend service.</summary>
<description>
The runner task owns the fixtures. Each run clears its observations and uses the same instances.
</description>
*)
METHOD PROTECTED ExecuteTest
VAR
	message : TOF_Core.ERROR_MESSAGE := "delivery probe";
	failuresBefore : ULINT;
END_VAR
IF NOT _QueueConfigured THEN
	_QueueConfigured := _Queue.Configure(backend := _Backend);
END_IF

Assert.ThatBool(actual := _QueueConfigured, message := "Queue must bind to its capture backend").IsTrue();

IF NOT _QueueConfigured THEN
	RETURN;
END_IF

Assert.ThatBool(
	actual := _Queue.PendingMessageCount = 0,
	message := "Scenario must start with an empty queue"
).IsTrue();

failuresBefore := _Queue.FailedDeliveryCount;
_Queue.Execute();
Assert.ThatBool(actual := _Backend.ExecuteCount = 1, message := "Empty queue must still service the backend").IsTrue();
_Backend.DeliveryBehavior := LOGGER_DELIVERY_BEHAVIOR.REFUSE;
Assert.ThatBool(
	actual := _Queue.TryLogMessage(category := TOF_Core.LOG_CATEGORY.ERROR, message := message),
	message := "First refusal probe must be admitted"
).IsTrue();
Assert.ThatBool(
	actual := _Queue.TryLogMessage(category := TOF_Core.LOG_CATEGORY.ERROR, message := message),
	message := "Second refusal probe must be admitted"
).IsTrue();
_Queue.Execute();
Assert.ThatBool(
	actual := _Queue.FailedDeliveryCount = failuresBefore + 2,
	message := "Refused attempts must be counted once each"
).IsTrue();
_Backend.DeliveryBehavior := LOGGER_DELIVERY_BEHAVIOR.THROW_EXCEPTION;
Assert.ThatBool(
	actual := _Queue.TryLogMessage(category := TOF_Core.LOG_CATEGORY.ERROR, message := message),
	message := "Delivery-exception probe must be admitted"
).IsTrue();
_Queue.Execute();
Assert.ThatBool(
	actual := _Queue.FailedDeliveryCount = failuresBefore + 3,
	message := "A hostile delivery exception must be contained and counted"
).IsTrue();
_Backend.DeliveryBehavior := LOGGER_DELIVERY_BEHAVIOR.ACCEPT;
_Backend.ThrowOnExecute := TRUE;
Assert.ThatBool(
	actual := _Queue.TryLogMessage(category := TOF_Core.LOG_CATEGORY.INFORMATION, message := message),
	message := "Record must be admitted while the backend Execute fault is armed"
).IsTrue();
_Queue.Execute();
_Backend.ThrowOnExecute := FALSE;
_Queue.Execute();
Assert.ThatBool(
	actual := _Backend.AttemptCount = 4,
	message := "Every dequeued record must have exactly one attempt"
).IsTrue();
Assert.ThatBool(
	actual := _Backend.CapturedCount = 1,
	message := "Normal delivery must resume after the nonfatal faults"
).IsTrue();
Assert.ThatBool(
	actual := _Backend.ExecuteCount = 5,
	message := "Execute faults must not prevent later service calls"
).IsTrue();
Assert.ThatBool(
	actual := _Queue.FailedDeliveryCount = failuresBefore + 3,
	message := "Backend Execute failure must not count as delivery failure"
).IsTrue();
Assert.ThatBool(actual := _Queue.PendingMessageCount = 0, message := "Failed records must not be retried").IsTrue();
END_METHOD

(*!
<summary>Clears capture observations and injected faults before each run.</summary>
*)
METHOD PROTECTED BeforeTest
_Backend.ResetCapture();
END_METHOD

//! <summary>Borrows the concrete class name for the instance lifetime. Callers must not modify it.</summary>
{attribute 'monitoring' := 'call'}
PROPERTY ClassName : REFERENCE TO STRING
GET
ClassName REF= _ClassName;
END_GET
END_PROPERTY

//! <summary>Borrows the compiler-initialized namespace. Callers must not modify it.</summary>
{attribute 'monitoring' := 'call'}
PROPERTY NamespaceName : REFERENCE TO STRING
GET
NamespaceName REF= CurrentNamespace.Name;
END_GET
END_PROPERTY

//! <summary>Reports the complete instance size in bytes, excluding separately allocated storage.</summary>
{attribute 'monitoring' := 'call'}
PROPERTY SelfSize : ULINT
GET
SelfSize := XSIZEOF(THIS^);
END_GET
END_PROPERTY

END_FUNCTION_BLOCK

// ---- Tests/Loggers/LoggerFormatterFailureTest.TcPOU
(*
SPDX-FileCopyrightText: c 2026 Oleksandr Tiutyk <trofimich@gmail.com>
SPDX-License-Identifier: MIT
License: https://opensource.org/license/mit
*)

(*!
<summary>Checks that all three logger types contain an exception raised by the message formatter.</summary>
<description>
The runner task owns the fixtures. Each run clears its observations and uses the same instances. The file
logger remains idle in INITIAL without cyclic service.
</description>
*)

{attribute 'no_assign'}
{attribute 'no_explicit_call' := 'do not call this function block directly'}
FUNCTION_BLOCK LoggerFormatterFailureTest EXTENDS TOF_Testing.SingleCycleTest
VAR_STAT
	{attribute 'hide'}
	_ClassName : STRING := __POUNAME();
END_VAR
VAR
	_Queue : TOF_Loggers.QueuedLogger;
	_Backend : LoggerCaptureBackend;
	_EventLogger : TOF_Loggers.EventLogger(
		debugEventType := TC_EVENTS.OpenFrameworkLoggerEventClass.DebugEvent,
		informationEventType := TC_EVENTS.OpenFrameworkLoggerEventClass.InformationEvent,
		warningEventType := TC_EVENTS.OpenFrameworkLoggerEventClass.WarningEvent,
		errorEventType := TC_EVENTS.OpenFrameworkLoggerEventClass.ErrorEvent,
		criticalErrorEventType := TC_EVENTS.OpenFrameworkLoggerEventClass.CriticalErrorEvent
	);
	_FileLogger : TOF_Loggers.SimpleTextFileLogger(
		directoryPath := '',
		logFilePrefix := 'Log',
		maxRecordsPerFile := 1,
		directoryPathType := Tc2_System.E_OpenPath.PATH_GENERIC,
		timeout := T#2S,
		amsNetId := ''
	);
	_Formatter : ThrowingGetMessageException;
	_QueueConfigured : BOOL;
END_VAR

(*!
<summary>Checks that all three logger types contain an exception raised by the message formatter.</summary>
<description>
The runner task owns the fixtures. Each run clears its observations and uses the same instances. The file
logger remains idle in INITIAL without cyclic service.
</description>
*)
METHOD PROTECTED ExecuteTest
VAR
	formatCallsBefore : UDINT;
END_VAR
IF NOT _QueueConfigured THEN
	_QueueConfigured := _Queue.Configure(backend := _Backend);
END_IF

Assert.ThatBool(actual := _QueueConfigured, message := "Queue must bind to its capture backend").IsTrue();

IF NOT _QueueConfigured THEN
	RETURN;
END_IF

Assert.ThatBool(
	actual := _Queue.PendingMessageCount = 0,
	message := "Scenario must start with an empty queue"
).IsTrue();
formatCallsBefore := _Formatter.MessageReadCount;
Assert.ThatBool(
	actual := _Queue.TryLogException(exception := _Formatter, severity := TOF_Core.ERROR_SEVERITY.ERROR),
	message := "Queued logger must contain a throwing formatter"
).IsFalse();
Assert.ThatUDInt(
	actual := _Formatter.MessageReadCount,
	message := "Queued logger must reach the throwing formatter"
).ToBe(expected := formatCallsBefore + 1);

formatCallsBefore := _Formatter.MessageReadCount;
Assert.ThatBool(
	actual := _FileLogger.TryLogException(exception := _Formatter, severity := TOF_Core.ERROR_SEVERITY.ERROR),
	message := "File logger must contain a throwing formatter before admission"
).IsFalse();
Assert.ThatUDInt(
	actual := _Formatter.MessageReadCount,
	message := "File logger must reach the throwing formatter"
).ToBe(expected := formatCallsBefore + 1);

formatCallsBefore := _Formatter.MessageReadCount;
Assert.ThatBool(
	actual := _EventLogger.TryLogException(exception := _Formatter, severity := TOF_Core.ERROR_SEVERITY.ERROR),
	message := "Event logger must contain a throwing formatter before native send"
).IsFalse();
Assert.ThatUDInt(
	actual := _Formatter.MessageReadCount,
	message := "Event logger must reach the throwing formatter"
).ToBe(expected := formatCallsBefore + 1);

Assert.ThatBool(
	actual := _Queue.PendingMessageCount = 0,
	message := "Failed formatting must not enqueue a record"
).IsTrue();
Assert.ThatBool(actual := _FileLogger.Busy, message := "INITIAL must still report pending initialization").IsTrue();
Assert.ThatBool(
	actual := _FileLogger.State = TOF_Loggers.SIMPLE_TEXT_FILE_LOGGER_STATE.INITIAL,
	message := "A formatting refusal must leave the file logger in INITIAL"
).IsTrue();
END_METHOD

(*!
<summary>Clears capture observations and injected faults before each run.</summary>
*)
METHOD PROTECTED BeforeTest
_Backend.ResetCapture();
END_METHOD

//! <summary>Borrows the concrete class name for the instance lifetime. Callers must not modify it.</summary>
{attribute 'monitoring' := 'call'}
PROPERTY ClassName : REFERENCE TO STRING
GET
ClassName REF= _ClassName;
END_GET
END_PROPERTY

//! <summary>Borrows the compiler-initialized namespace. Callers must not modify it.</summary>
{attribute 'monitoring' := 'call'}
PROPERTY NamespaceName : REFERENCE TO STRING
GET
NamespaceName REF= CurrentNamespace.Name;
END_GET
END_PROPERTY

//! <summary>Reports the complete instance size in bytes, excluding separately allocated storage.</summary>
{attribute 'monitoring' := 'call'}
PROPERTY SelfSize : ULINT
GET
SelfSize := XSIZEOF(THIS^);
END_GET
END_PROPERTY

END_FUNCTION_BLOCK

// ---- Tests/Loggers/LoggerMetadataAndRecordLimitTest.TcPOU
(*
SPDX-FileCopyrightText: c 2026 Oleksandr Tiutyk <trofimich@gmail.com>
SPDX-License-Identifier: MIT
License: https://opensource.org/license/mit
*)

(*!
<summary>Checks logger metadata and rejection of a zero file record limit.</summary>
<description>
Use in the runner task. The first run exercises INITIAL to FAILED; later runs check the retained terminal state.
</description>
*)

{attribute 'no_assign'}
{attribute 'no_explicit_call' := 'do not call this function block directly'}
FUNCTION_BLOCK LoggerMetadataAndRecordLimitTest EXTENDS TOF_Testing.SingleCycleTest
VAR_STAT
	{attribute 'hide'}
	_ClassName : STRING := __POUNAME();
END_VAR
VAR
	_Queue : TOF_Loggers.QueuedLogger;
	_EventLogger : TOF_Loggers.EventLogger(
		debugEventType := TC_EVENTS.OpenFrameworkLoggerEventClass.DebugEvent,
		informationEventType := TC_EVENTS.OpenFrameworkLoggerEventClass.InformationEvent,
		warningEventType := TC_EVENTS.OpenFrameworkLoggerEventClass.WarningEvent,
		errorEventType := TC_EVENTS.OpenFrameworkLoggerEventClass.ErrorEvent,
		criticalErrorEventType := TC_EVENTS.OpenFrameworkLoggerEventClass.CriticalErrorEvent
	);
	_FileLogger : TOF_Loggers.SimpleTextFileLogger(
		directoryPath := '',
		logFilePrefix := 'Log',
		maxRecordsPerFile := 0,
		directoryPathType := Tc2_System.E_OpenPath.PATH_GENERIC,
		timeout := T#2S,
		amsNetId := ''
	);
	_Formatter : ThrowingGetMessageException;
	_InitialConfigurationChecked : BOOL;
END_VAR

(*!
<summary>Checks logger metadata and rejection of a zero file record limit.</summary>
<description>
Use in the runner task. The first run exercises INITIAL to FAILED; later runs check the retained terminal state.
</description>
*)
METHOD PROTECTED ExecuteTest
VAR
	error : TOF_Core.ERROR;
	message : TOF_Core.ERROR_MESSAGE := "must be refused";
	formatCallsBefore : UDINT;
END_VAR
Assert.ThatBool(
	actual := _Queue.ClassName = 'QueuedLogger',
	message := "Queue metadata must identify its concrete type"
).IsTrue();
Assert.ThatBool(
	actual := _EventLogger.ClassName = 'EventLogger',
	message := "Event metadata must identify its concrete type"
).IsTrue();
Assert.ThatBool(
	actual := _FileLogger.ClassName = 'SimpleTextFileLogger',
	message := "File metadata must identify its concrete type"
).IsTrue();
Assert.ThatBool(
	actual := _FileLogger.NamespaceName = 'TOF_Loggers',
	message := "File namespace must remain unchanged"
).IsTrue();
Assert.ThatBool(
	actual := _FileLogger.SelfSize = XSIZEOF(_FileLogger),
	message := "Size must describe the concrete instance"
).IsTrue();
Assert.ThatBool(actual := _FileLogger.Timeout = T#2S, message := "Configured native timeout must be retained").IsTrue();
IF NOT _InitialConfigurationChecked THEN
	Assert.ThatBool(
		actual := _FileLogger.State = TOF_Loggers.SIMPLE_TEXT_FILE_LOGGER_STATE.INITIAL,
		message := "The invalid configuration must be tested before the first Execute"
	).IsTrue();
END_IF

error.SetMessage(message := "invalid limit error");
formatCallsBefore := _Formatter.MessageReadCount;
Assert.ThatBool(
	actual := _FileLogger.TryLogMessage(category := TOF_Core.LOG_CATEGORY.INFORMATION, message := message),
	message := "Zero record limit must refuse plain admission"
).IsFalse();
Assert.ThatBool(
	actual := _FileLogger.TryLogError(error := error),
	message := "Zero record limit must refuse errors"
).IsFalse();
Assert.ThatBool(
	actual := _FileLogger.TryLogException(exception := _Formatter, severity := TOF_Core.ERROR_SEVERITY.ERROR),
	message := "Zero record limit must refuse before formatting"
).IsFalse();
Assert.ThatUDInt(
	actual := _Formatter.MessageReadCount,
	message := "The invalid configuration must refuse before reading the exception"
).ToBe(expected := formatCallsBefore);

_FileLogger.Execute();
_InitialConfigurationChecked := TRUE;
Assert.ThatBool(
	actual := _FileLogger.State = TOF_Loggers.SIMPLE_TEXT_FILE_LOGGER_STATE.FAILED,
	message := "Zero record limit must fail before attempting the deliberately empty directory"
).IsTrue();
Assert.ThatBool(
	actual := _FileLogger.ErrorMessage = "MaxRecordsPerFile must be greater than zero.",
	message := "Configuration diagnostic must explain the invalid record limit"
).IsTrue();
Assert.ThatBool(
	actual := _FileLogger.Busy,
	message := "No native cleanup may remain after the configuration failure"
).IsFalse();
Assert.ThatBool(actual := _FileLogger.Start(), message := "FAILED must remain terminal").IsFalse();
END_METHOD

//! <summary>Borrows the concrete class name for the instance lifetime. Callers must not modify it.</summary>
{attribute 'monitoring' := 'call'}
PROPERTY ClassName : REFERENCE TO STRING
GET
ClassName REF= _ClassName;
END_GET
END_PROPERTY

//! <summary>Borrows the compiler-initialized namespace. Callers must not modify it.</summary>
{attribute 'monitoring' := 'call'}
PROPERTY NamespaceName : REFERENCE TO STRING
GET
NamespaceName REF= CurrentNamespace.Name;
END_GET
END_PROPERTY

//! <summary>Reports the complete instance size in bytes, excluding separately allocated storage.</summary>
{attribute 'monitoring' := 'call'}
PROPERTY SelfSize : ULINT
GET
SelfSize := XSIZEOF(THIS^);
END_GET
END_PROPERTY

END_FUNCTION_BLOCK

// ---- Tests/Loggers/LoggerTaskDiagnosticsTest.TcPOU
(*
SPDX-FileCopyrightText: c 2026 Oleksandr Tiutyk <trofimich@gmail.com>
SPDX-License-Identifier: MIT
License: https://opensource.org/license/mit
*)

(*!
<summary>Checks that explicit task diagnostics bypass the reject-all filter without servicing the destination.</summary>
<description>
The runner task owns the fixtures. Each run clears its observations and uses the same instances. An explicit
per-test reject-all filter is installed only within one synchronous call.
</description>
*)

{attribute 'no_assign'}
{attribute 'no_explicit_call' := 'do not call this function block directly'}
FUNCTION_BLOCK LoggerTaskDiagnosticsTest EXTENDS TOF_Testing.SingleCycleTest
VAR_STAT
	{attribute 'hide'}
	_ClassName : STRING := __POUNAME();
END_VAR
VAR
	_Task : LoggerTaskProbe(name := "diagnostic route probe");
	_Backend : LoggerCaptureBackend;
	_Filter : LogFilter;
END_VAR

(*!
<summary>Checks that explicit task diagnostics bypass the reject-all filter without servicing the destination.</summary>
<description>
The runner task owns the fixtures. Each run clears its observations and uses the same instances. An explicit
per-test reject-all filter is installed only within one synchronous call.
</description>
*)
METHOD PROTECTED ExecuteTest
VAR
	savedFilter : TOF_Core.ILogFilter;
	escaped : BOOL;
END_VAR
savedFilter := TOF_Core.LogManager.Filter;
TOF_Core.LogManager.Filter := _Filter;

__TRY
	_Task.DiagnosticLogger := _Backend;
	Assert.ThatBool(actual := _Task.Start(), message := "Prepared probe must start").IsTrue();
	Assert.ThatUInt(actual := _Backend.CapturedCount, message := "Start must emit one RUNNING diagnostic").ToBe(
		expected := 1
	);

	_Task.Execute();
	Assert.ThatBool(actual := _Task.State.Stopped, message := "Probe must complete without native I/O").IsTrue();
	Assert.ThatUInt(actual := _Backend.CapturedCount, message := "Execute must add one STOPPED diagnostic").ToBe(
		expected := 2
	);

	Assert.ThatBool(actual := _Task.Reset(), message := "Stopped probe must reset").IsTrue();
	Assert.ThatBool(
		actual := _Backend.CapturedCount = 3,
		message := "Reset must add one READY diagnostic"
	).IsTrue();
	Assert.ThatBool(
		actual := _Backend.ExecuteCount = 0,
		message := "Task must not take ownership of diagnostic execution"
	).IsTrue();
__CATCH
	escaped := TRUE;
__ENDTRY

TOF_Core.LogManager.Filter := savedFilter;
Assert.ThatBool(actual := escaped, message := "The diagnostic scenario must return normally").IsFalse();
END_METHOD

(*!
<summary>Clears diagnostic observations before running the probe again.</summary>
*)
METHOD PROTECTED BeforeTest
_Backend.ResetCapture();
END_METHOD

//! <summary>Borrows the concrete class name for the instance lifetime. Callers must not modify it.</summary>
{attribute 'monitoring' := 'call'}
PROPERTY ClassName : REFERENCE TO STRING
GET
ClassName REF= _ClassName;
END_GET
END_PROPERTY

//! <summary>Borrows the compiler-initialized namespace. Callers must not modify it.</summary>
{attribute 'monitoring' := 'call'}
PROPERTY NamespaceName : REFERENCE TO STRING
GET
NamespaceName REF= CurrentNamespace.Name;
END_GET
END_PROPERTY

//! <summary>Reports the complete instance size in bytes, excluding separately allocated storage.</summary>
{attribute 'monitoring' := 'call'}
PROPERTY SelfSize : ULINT
GET
SelfSize := XSIZEOF(THIS^);
END_GET
END_PROPERTY

END_FUNCTION_BLOCK

// ---- Tests/Loggers/LoggerTaskProbe.TcPOU
(*
SPDX-FileCopyrightText: © 2026 Oleksandr Tiutyk <trofimich@gmail.com>
SPDX-License-Identifier: MIT
License: https://opensource.org/license/mit
*)
(*!
<summary>Completes one task cycle to expose internal lifecycle diagnostics.</summary>
<description>
The inherited DiagnosticLogger is configured by the owning regression before Start; no native I/O occurs.
</description>
*)

{attribute 'no_explicit_call' := 'do not call this function block directly'}
FUNCTION_BLOCK LoggerTaskProbe EXTENDS TOF_Tasks.Task
VAR_STAT
	//! <summary>Concrete type metadata available during base initialization.</summary>
	_ClassName : STRING := __POUNAME();
END_VAR

(*!
<summary>Borrows the concrete fixture type name.</summary>
<description>
Returns initialized static metadata; do not modify the referenced string.
</description>
*)
{attribute 'monitoring' := 'call'}
PROPERTY ClassName : REFERENCE TO STRING
GET
ClassName REF= _ClassName;
END_GET
END_PROPERTY

(*!
<summary>Borrows the test namespace.</summary>
<description>
Returns compiler-initialized library storage without ownership transfer.
</description>
*)
{attribute 'monitoring' := 'call'}
PROPERTY NamespaceName : REFERENCE TO STRING
GET
NamespaceName REF= CurrentNamespace.Name;
END_GET
END_PROPERTY

(*!
<summary>Completes immediately without external resources.</summary>
*)
METHOD PROTECTED OnRunning
VAR_OUTPUT
	processingState : TOF_Tasks.TASK_PROCESSING_STATE;
END_VAR
VAR_IN_OUT
	stopReasonMessage : TOF_Core.ERROR_MESSAGE;
END_VAR
processingState := TOF_Tasks.TASK_PROCESSING_STATE.DONE;
END_METHOD

(*!
<summary>Reports the concrete fixture size in bytes.</summary>
*)
{attribute 'monitoring' := 'call'}
PROPERTY SelfSize : ULINT
GET
SelfSize := XSIZEOF(THIS^);
END_GET
END_PROPERTY

END_FUNCTION_BLOCK

// ---- LogFilter.TcPOU
(*
SPDX-FileCopyrightText: © 2026 Oleksandr Tiutyk <trofimich@gmail.com>
SPDX-License-Identifier: MIT
License: https://opensource.org/license/mit
*)

(*!
<summary>Suppresses test log output and optionally simulates reuse of a native diagnostic during logging.</summary>
<description>Probe state belongs to the calling cyclic task. The filter never retains the borrowed exception.</description>
*)

{attribute 'no_explicit_call' := 'do not call this function block directly'}
FUNCTION_BLOCK LogFilter EXTENDS TOF_Core.Object IMPLEMENTS TOF_Core.ILogFilter
VAR
	_SecondaryExceptionPending : ARRAY [1..TOF_Core.System.TASK_COUNT] OF BOOL;
END_VAR
VAR_STAT
	//! <summary>Class name shared by all instances of this function block.</summary>
	{attribute 'hide'} 
	_ClassName : STRING := __POUNAME();
END_VAR

{attribute 'monitoring' := 'call'}
PROPERTY ClassName : REFERENCE TO STRING
GET
ClassName REF= _ClassName;
END_GET
END_PROPERTY

{attribute 'monitoring' := 'call'}
PROPERTY NamespaceName : REFERENCE TO STRING
GET
NamespaceName REF= CurrentNamespace.Name;
END_GET
END_PROPERTY

{attribute 'monitoring' := 'call'}
PROPERTY SelfSize : ULINT
GET
SelfSize := XSIZEOF(THIS^);
END_GET
END_PROPERTY

(*! <summary>Consumes any armed secondary diagnostic in this task and suppresses the log entry.</summary> *)
METHOD ShouldLog : BOOL
VAR_IN_OUT CONSTANT
	category : TOF_Core.LOG_CATEGORY;
	topics : ARRAY [*] OF WSTRING;		
END_VAR
VAR
	taskIndex : DINT;
END_VAR
taskIndex := TOF_Core.System.GetCurrentTaskIndex();

IF taskIndex >= 1
	AND_THEN taskIndex <= TOF_Core.System.TASK_COUNT
	AND_THEN _SecondaryExceptionPending[taskIndex]
THEN
	_SecondaryExceptionPending[taskIndex] := FALSE;
	TOF_Core.ExceptionManager.GetLastException(
		exceptionCode := __SYSTEM.ExceptionCode.RTSEXCPT_ACCESS_VIOLATION,
		catchPointNamespaceName := NamespaceName,
		catchPointPOUName := __POUNAME(),
		catchPointPosition := __POSITION()
	);
END_IF

ShouldLog := FALSE;
END_METHOD

(*!
<summary>Enables or cancels one simulated secondary native diagnostic in the calling test task.</summary>
<description>Each cyclic task owns its slot. Other tasks keep their configured filter behavior.</description>
<param name="enabled">TRUE arms the next logging callback. FALSE cancels a pending probe.</param>
*)
METHOD SetSecondaryExceptionProbe
VAR_INPUT
	enabled : BOOL;
END_VAR
VAR
	taskIndex : DINT;
END_VAR
taskIndex := TOF_Core.System.GetCurrentTaskIndex();

IF taskIndex >= 1 AND_THEN taskIndex <= TOF_Core.System.TASK_COUNT THEN
	_SecondaryExceptionPending[taskIndex] := enabled;
END_IF
END_METHOD

END_FUNCTION_BLOCK

// ---- Tests/Loggers/QueuedLoggerAggregateTest.TcPOU
(*
SPDX-FileCopyrightText: c 2026 Oleksandr Tiutyk <trofimich@gmail.com>
SPDX-License-Identifier: MIT
License: https://opensource.org/license/mit
*)

(*!
<summary>Checks aggregate ordering, copied diagnostic text and partial admission when the queue fills.</summary>
<description>
The queue and capture belong to the runner task. Clears borrowed exception references before leaving the call.
</description>
*)

{attribute 'no_assign'}
{attribute 'no_explicit_call' := 'do not call this function block directly'}
FUNCTION_BLOCK QueuedLoggerAggregateTest EXTENDS TOF_Testing.SingleCycleTest
VAR_STAT
	{attribute 'hide'}
	_ClassName : STRING := __POUNAME();
END_VAR
VAR
	_Queue : TOF_Loggers.QueuedLogger;
	_Backend : LoggerCaptureBackend;
	_Aggregate : TOF_Core.AggregateException;
	_QueueConfigured : BOOL;
END_VAR

(*!
<summary>Checks aggregate ordering, copied diagnostic text and partial admission when the queue fills.</summary>
<description>
The queue and capture belong to the runner task. Clears borrowed exception references before leaving the call.
</description>
*)
METHOD PROTECTED ExecuteTest
VAR
	firstCause : TOF_Core.IException;
	secondCause : TOF_Core.IException;
	exceptionCode : __SYSTEM.ExceptionCode;
	record : LOGGER_CAPTURED_MESSAGE;
	firstMessage : TOF_Core.ERROR_MESSAGE;
	secondMessage : TOF_Core.ERROR_MESSAGE;
	escaped : BOOL;
	number : ULINT;
	i : DINT;
END_VAR
IF NOT _QueueConfigured THEN
	_QueueConfigured := _Queue.Configure(backend := _Backend);
END_IF

Assert.ThatBool(actual := _QueueConfigured, message := "Queue must bind to its capture backend").IsTrue();

IF NOT _QueueConfigured THEN
	RETURN;
END_IF

Assert.ThatBool(
	actual := _Queue.PendingMessageCount = 0,
	message := "Scenario must start with an empty queue"
).IsTrue();

__TRY

	__TRY
		TOF_Core.Exceptions.ThrowStandard(
			sourceNamespaceName := NamespaceName,
			sourceClassName := ClassName,
			sourcePOUName := __POUNAME(),
			sourcePosition := __POSITION(),
			message := "first aggregate cause"
		);
	__CATCH(exceptionCode)
		firstCause := TOF_Core.ExceptionManager.GetLastException(
			exceptionCode := exceptionCode,
			catchPointNamespaceName := NamespaceName,
			catchPointPOUName := __POUNAME(),
			catchPointPosition := __POSITION()
		);
	__ENDTRY

	__TRY
		TOF_Core.Exceptions.ThrowStandard(
			sourceNamespaceName := NamespaceName,
			sourceClassName := ClassName,
			sourcePOUName := __POUNAME(),
			sourcePosition := __POSITION(),
			message := "second aggregate cause"
		);
	__CATCH(exceptionCode)
		secondCause := TOF_Core.ExceptionManager.GetLastException(
			exceptionCode := exceptionCode,
			catchPointNamespaceName := NamespaceName,
			catchPointPOUName := __POUNAME(),
			catchPointPosition := __POSITION()
		);
	__ENDTRY

	Assert.ThatBool(
		actual := firstCause <> 0 AND_THEN secondCause <> 0 AND_THEN firstCause <> secondCause,
		message := "The two injected failures must provide distinct live cause objects"
	).IsTrue();

	IF firstCause = 0 OR_ELSE secondCause = 0 THEN
		RETURN;
	END_IF

	_Aggregate.AddInnerException(innerException := firstCause);
	_Aggregate.AddInnerException(innerException := secondCause);
	firstMessage := firstCause.GetMessage(
		showSource := TRUE,
		timestampDisplayMode := TOF_Core.TIMESTAMP_DISPLAY_MODE.LOCAL
	);
	secondMessage := secondCause.GetMessage(
		showSource := TRUE,
		timestampDisplayMode := TOF_Core.TIMESTAMP_DISPLAY_MODE.LOCAL
	);
	Assert.ThatBool(actual := firstMessage <> secondMessage, message := "Cause texts must be distinct").IsTrue();

	number := 73;
	Assert.ThatBool(
		actual := _Queue.TryLogException(
			exception := _Aggregate,
			severity := TOF_Core.ERROR_SEVERITY.ERROR,
			messageNumber := number
		),
		message := "Both aggregate causes must be accepted in order"
	).IsTrue();

	number := 99;
	_Queue.Execute();
	Assert.ThatUInt(actual := _Backend.CapturedCount, message := "Aggregate must deliver two records").ToBe(expected := 2);
	record := _Backend.RecordAt(index := 0);
	Assert.ThatBool(actual := record.Message = firstMessage, message := "First cause must be delivered first").IsTrue();
	Assert.ThatBool(
		actual := record.Category = TOF_Core.LOG_CATEGORY.ERROR AND_THEN record.HasMessageNumber
			AND_THEN record.MessageNumber = 73,
		message := "First cause must retain its category and copied request number"
	).IsTrue();

	record := _Backend.RecordAt(index := 1);
	Assert.ThatBool(
		actual := record.Message = secondMessage,
		message := "Second cause must be delivered second"
	).IsTrue();
	Assert.ThatBool(
		actual := record.Category = TOF_Core.LOG_CATEGORY.ERROR AND_THEN record.HasMessageNumber
			AND_THEN record.MessageNumber = 73,
		message := "Second cause must retain its category and copied request number"
	).IsTrue();

	FOR i := 1 TO TO_DINT(TOF_Loggers.Parameters.QUEUED_LOGGER_CAPACITY) - 1 DO
		Assert.ThatBool(
			actual := _Queue.TryLogMessage(category := TOF_Core.LOG_CATEGORY.DEBUG, message := "reserved queue slot"),
			message := "The reserved slot must be filled"
		).IsTrue();
	END_FOR

	number := 74;
	Assert.ThatBool(
		actual := _Queue.TryLogException(
			exception := _Aggregate,
			severity := TOF_Core.ERROR_SEVERITY.ERROR,
			messageNumber := number
		),
		message := "An aggregate with only one free slot must report partial admission"
	).IsFalse();

	_Aggregate.Clear();
	_Queue.Execute();
	Assert.ThatUInt(actual := _Backend.CapturedCount, message := "Exactly one additional cause must be delivered").ToBe(
		expected := TOF_Loggers.Parameters.QUEUED_LOGGER_CAPACITY + 2
	);
	record := _Backend.RecordAt(index := TOF_Loggers.Parameters.QUEUED_LOGGER_CAPACITY + 1);
	Assert.ThatBool(
		actual := record.Message = firstMessage,
		message := "Accepted text must survive aggregate Clear"
	).IsTrue();
	Assert.ThatBool(
		actual := record.HasMessageNumber AND_THEN record.MessageNumber = 74,
		message := "The partially admitted cause must retain this request number"
	).IsTrue();
	Assert.ThatBool(
		actual := _Queue.PendingMessageCount = 0,
		message := "All partially admitted entries must drain"
	).IsTrue();
__CATCH
	escaped := TRUE;
__ENDTRY

_Aggregate.Clear();
Assert.ThatBool(actual := escaped, message := "The aggregate scenario must return normally").IsFalse();
END_METHOD

(*!
<summary>Clears capture observations and injected faults before each run.</summary>
*)
METHOD PROTECTED BeforeTest
_Backend.ResetCapture();
END_METHOD

//! <summary>Borrows the concrete class name for the instance lifetime. Callers must not modify it.</summary>
{attribute 'monitoring' := 'call'}
PROPERTY ClassName : REFERENCE TO STRING
GET
ClassName REF= _ClassName;
END_GET
END_PROPERTY

//! <summary>Borrows the compiler-initialized namespace. Callers must not modify it.</summary>
{attribute 'monitoring' := 'call'}
PROPERTY NamespaceName : REFERENCE TO STRING
GET
NamespaceName REF= CurrentNamespace.Name;
END_GET
END_PROPERTY

//! <summary>Reports the complete instance size in bytes, excluding separately allocated storage.</summary>
{attribute 'monitoring' := 'call'}
PROPERTY SelfSize : ULINT
GET
SelfSize := XSIZEOF(THIS^);
END_GET
END_PROPERTY

END_FUNCTION_BLOCK

// ---- Tests/Loggers/CurrentTaskLoggerRoutingTest.TcPOU
(*
SPDX-FileCopyrightText: c 2026 Oleksandr Tiutyk <trofimich@gmail.com>
SPDX-License-Identifier: MIT
License: https://opensource.org/license/mit
*)

(*!
<summary>Checks task destination assignment, default reset, queued diagnostics and service failure containment.</summary>
<description>
Owns the queue and captures in the runner task. The task destination, shared filter and numbering are restored
within the same call. No other task may log while the shared settings are temporarily changed.
</description>
*)

{attribute 'no_assign'}
{attribute 'no_explicit_call' := 'do not call this function block directly'}
FUNCTION_BLOCK CurrentTaskLoggerRoutingTest EXTENDS TOF_Testing.SingleCycleTest
VAR_STAT
	{attribute 'hide'}
	_ClassName : STRING := __POUNAME();
END_VAR
VAR
	_Backend : LoggerCaptureBackend;
	_Queue : TOF_Loggers.QueuedLogger;
	_QueueConfigured : BOOL;
END_VAR

(*!
<summary>Checks task destination assignment, default reset, queued diagnostics and service failure containment.</summary>
<description>
Owns the queue and captures in the runner task. The task destination, shared filter and numbering are restored
within the same call. No other task may log while the shared settings are temporarily changed.
</description>
*)
METHOD PROTECTED ExecuteTest
VAR
	backendLogger : TOF_Core.ILogger;
	savedLogger : TOF_Core.ILogger;
	defaultLogger : TOF_Core.ILogger;
	selectedLogger : TOF_Core.ILogger;
	savedFilter : TOF_Core.ILogFilter;
	savedFormat : TOF_Core.LOG_MESSAGE_NUMBER_FORMAT;
	error : TOF_Core.ERROR;
	message : TOF_Core.ERROR_MESSAGE := "current task destination";
	expectedError : TOF_Core.ERROR_MESSAGE;
	expectedException : TOF_Core.ERROR_MESSAGE;
	record : LOGGER_CAPTURED_MESSAGE;
	escaped : BOOL;
	exceptionCode : __SYSTEM.ExceptionCode;
	routedException : TOF_Core.IException;
END_VAR
IF NOT _QueueConfigured THEN
	_QueueConfigured := _Queue.Configure(backend := _Backend);
END_IF

Assert.ThatBool(actual := _QueueConfigured, message := "Queue must bind to its capture backend").IsTrue();

IF NOT _QueueConfigured THEN
	RETURN;
END_IF

Assert.ThatBool(
	actual := _Queue.PendingMessageCount = 0,
	message := "Scenario must start with an empty queue"
).IsTrue();

__TRY
	TOF_Core.Exceptions.ThrowStandard(
		sourceNamespaceName := NamespaceName,
		sourceClassName := ClassName,
		sourcePOUName := __POUNAME(),
		sourcePosition := __POSITION(),
		message := "current task exception"
	);
__CATCH(exceptionCode)
	routedException := TOF_Core.ExceptionManager.GetLastException(
		exceptionCode := exceptionCode,
		catchPointNamespaceName := NamespaceName,
		catchPointPOUName := __POUNAME(),
		catchPointPosition := __POSITION()
	);
__ENDTRY

Assert.ThatBool(actual := routedException <> 0, message := "The routing probe needs a live exception").IsTrue();

IF routedException = 0 THEN
	RETURN;
END_IF

savedLogger := TOF_Core.LogManager.CurrentTaskLogger;
savedFilter := TOF_Core.LogManager.Filter;
savedFormat := TOF_Core.LogManager.MessageNumberFormat;

__TRY
	TOF_Core.LogManager.Filter := 0;
	TOF_Core.LogManager.MessageNumberFormat := TOF_Core.LOG_MESSAGE_NUMBER_FORMAT.NONE;
	TOF_Core.LogManager.CurrentTaskLogger := 0;
	defaultLogger := TOF_Core.LogManager.CurrentTaskLogger;
	Assert.ThatBool(
		actual := defaultLogger <> 0,
		message := "Cyclic task must have a standard ADS destination"
	).IsTrue();
	TOF_Core.LogManager.CurrentTaskLogger := _Backend;
	selectedLogger := TOF_Core.LogManager.CurrentTaskLogger;
	backendLogger := _Backend;
	Assert.ThatBool(
		actual := selectedLogger = backendLogger,
		message := "Getter must return the task assignment"
	).IsTrue();
	Assert.ThatBool(
		actual := TOF_Core.LogManager.TryLogMessage(
			message := message,
			category := TOF_Core.LOG_CATEGORY.INFORMATION
		),
		message := "Manager must route text to the assigned backend"
	).IsTrue();
	TOF_Core.LogManager.ExecuteCurrentTaskLogger();
	Assert.ThatBool(
		actual := _Backend.CapturedCount = 1,
		message := "Assigned backend must receive the message"
	).IsTrue();
	Assert.ThatBool(
		actual := _Backend.ExecuteCount = 1,
		message := "Service must use the same task destination"
	).IsTrue();
	record := _Backend.RecordAt(index := 0);
	Assert.ThatBool(actual := record.Message = message, message := "Manager must preserve routed text").IsTrue();
	Assert.ThatBool(actual := record.HasMessageNumber, message := "NONE must omit the request number").IsFalse();

	TOF_Core.LogManager.CurrentTaskLogger := _Queue;
	error.SetMessage(message := "current task error");
	expectedError := error.ToString(
		sourceDisplayMode := TOF_Core.ERROR_SOURCE_DISPLAY_MODE.TOP_AND_ROOT,
		timestampDisplayMode := TOF_Core.TIMESTAMP_DISPLAY_MODE.LOCAL
	);
	expectedException := routedException.GetMessage(
		showSource := TRUE,
		timestampDisplayMode := TOF_Core.TIMESTAMP_DISPLAY_MODE.LOCAL
	);
	Assert.ThatBool(
		actual := TOF_Core.LogManager.TryLogMessage(
			message := message,
			category := TOF_Core.LOG_CATEGORY.INFORMATION
		),
		message := "Replacement queue must accept the manager message"
	).IsTrue();
	Assert.ThatBool(
		actual := TOF_Core.LogManager.TryLogError(error := error),
		message := "Manager must route errors to the replacement queue"
	).IsTrue();
	Assert.ThatBool(
		actual := TOF_Core.LogManager.TryLogException(
			exception := routedException,
			severity := TOF_Core.ERROR_SEVERITY.ERROR
		),
		message := "Manager must route exceptions to the replacement queue"
	).IsTrue();
	Assert.ThatBool(actual := _Backend.CapturedCount = 1, message := "Admission must not bypass the queue").IsTrue();
	Assert.ThatBool(
		actual := _Queue.PendingMessageCount = 3,
		message := "All three manager methods must use the queue"
	).IsTrue();
	TOF_Core.LogManager.ExecuteCurrentTaskLogger();
	Assert.ThatBool(
		actual := _Backend.ExecuteCount = 2,
		message := "Manager service must advance the queue backend once"
	).IsTrue();
	Assert.ThatBool(
		actual := _Backend.CapturedCount = 4,
		message := "Service must deliver all queued manager records"
	).IsTrue();
	Assert.ThatBool(
		actual := _Queue.PendingMessageCount = 0,
		message := "Owner service must drain the queued records"
	).IsTrue();
	record := _Backend.RecordAt(index := 1);
	Assert.ThatBool(actual := record.Message = message, message := "Queue must preserve the routed message").IsTrue();
	Assert.ThatBool(
		actual := record.HasMessageNumber,
		message := "Queue must preserve the absent request number"
	).IsFalse();

	record := _Backend.RecordAt(index := 2);
	Assert.ThatBool(
		actual := record.Message = expectedError,
		message := "Error delivery must preserve formatted text"
	).IsTrue();
	record := _Backend.RecordAt(index := 3);
	Assert.ThatBool(
		actual := record.Message = expectedException,
		message := "Exception delivery must preserve formatted text"
	).IsTrue();
	TOF_Core.LogManager.CurrentTaskLogger := 0;
	selectedLogger := TOF_Core.LogManager.CurrentTaskLogger;
	Assert.ThatBool(
		actual := selectedLogger = defaultLogger,
		message := "Zero must restore the same task ADS instance"
	).IsTrue();
	TOF_Core.LogManager.ExecuteCurrentTaskLogger();
	Assert.ThatBool(
		actual := _Backend.ExecuteCount = 2,
		message := "Reset must stop servicing the replaced backend"
	).IsTrue();
	TOF_Core.LogManager.CurrentTaskLogger := _Backend;
	_Backend.ThrowOnExecute := TRUE;
	TOF_Core.LogManager.ExecuteCurrentTaskLogger();
	Assert.ThatBool(
		actual := _Backend.ExecuteCount = 3,
		message := "A hostile Execute must be attempted once"
	).IsTrue();
	Assert.ThatBool(
		actual := _Backend.CapturedCount = 4,
		message := "Execute failure diagnostics must bypass the task route"
	).IsTrue();
	_Backend.ThrowOnExecute := FALSE;
	_Backend.DeliveryBehavior := LOGGER_DELIVERY_BEHAVIOR.THROW_EXCEPTION;
	Assert.ThatBool(
		actual := TOF_Core.LogManager.TryLogMessage(
			message := message,
			category := TOF_Core.LOG_CATEGORY.INFORMATION
		),
		message := "Manager must contain a hostile task logger TryLog exception"
	).IsFalse();
	Assert.ThatUInt(actual := _Backend.AttemptCount, message := "Hostile TryLog must reach the backend once").ToBe(
		expected := 5
	);
__CATCH
	escaped := TRUE;
__ENDTRY

_Backend.ThrowOnExecute := FALSE;
_Backend.DeliveryBehavior := LOGGER_DELIVERY_BEHAVIOR.ACCEPT;
TOF_Core.LogManager.CurrentTaskLogger := savedLogger;
TOF_Core.LogManager.Filter := savedFilter;
TOF_Core.LogManager.MessageNumberFormat := savedFormat;
Assert.ThatBool(actual := escaped, message := "The task routing scenario must return normally").IsFalse();
END_METHOD

(*!
<summary>Clears capture observations and injected faults before each run.</summary>
*)
METHOD PROTECTED BeforeTest
_Backend.ResetCapture();
END_METHOD

//! <summary>Borrows the concrete class name for the instance lifetime. Callers must not modify it.</summary>
{attribute 'monitoring' := 'call'}
PROPERTY ClassName : REFERENCE TO STRING
GET
ClassName REF= _ClassName;
END_GET
END_PROPERTY

//! <summary>Borrows the compiler-initialized namespace. Callers must not modify it.</summary>
{attribute 'monitoring' := 'call'}
PROPERTY NamespaceName : REFERENCE TO STRING
GET
NamespaceName REF= CurrentNamespace.Name;
END_GET
END_PROPERTY

//! <summary>Reports the complete instance size in bytes, excluding separately allocated storage.</summary>
{attribute 'monitoring' := 'call'}
PROPERTY SelfSize : ULINT
GET
SelfSize := XSIZEOF(THIS^);
END_GET
END_PROPERTY

END_FUNCTION_BLOCK

// ---- Tests/Loggers/LoggerNonCyclicInitializationTest.TcPOU
(*
SPDX-FileCopyrightText: c 2026 Oleksandr Tiutyk <trofimich@gmail.com>
SPDX-License-Identifier: MIT
License: https://opensource.org/license/mit
*)

(*!
<summary>Asserts the non-cyclic FB_init probe and absence of an initialization logger assignment.</summary>
<description>
Captures initialization observations once and checks them in each cyclic run. The runner retains no logger alias.
</description>
*)

{attribute 'no_assign'}
{attribute 'no_explicit_call' := 'do not call this function block directly'}
FUNCTION_BLOCK LoggerNonCyclicInitializationTest EXTENDS TOF_Testing.SingleCycleTest
VAR_STAT
	{attribute 'hide'}
	_ClassName : STRING := __POUNAME();
END_VAR
VAR
	//! <summary>Records that initialization exercised a non-cyclic execution context.</summary>
	_InitializationContextObserved : BOOL;
	//! <summary>Records rejection without exceptions, counter changes or a published non-cyclic destination.</summary>
	_InitializationCallsRejected : BOOL;
	_InitializationLogger : TOF_Core.AdsLogger;
	_InitializationError : TOF_Core.ERROR;
	_InitializationException : TOF_Core.StandardException;
END_VAR

(*!
<summary>Asserts the non-cyclic FB_init probe and absence of an initialization logger assignment.</summary>
<description>
Captures initialization observations once and checks them in each cyclic run. The runner retains no logger alias.
</description>
*)
METHOD PROTECTED ExecuteTest
VAR
	currentLogger : TOF_Core.ILogger;
	initializationLogger : TOF_Core.ILogger;
END_VAR
Assert.ThatBool(
	actual := _InitializationContextObserved,
	message := "FB_init must exercise a non-cyclic context"
).IsTrue();
Assert.ThatBool(
	actual := _InitializationCallsRejected,
	message := "Non-cyclic calls must return defaults without logging or changing counters"
).IsTrue();
currentLogger := TOF_Core.LogManager.CurrentTaskLogger;
initializationLogger := _InitializationLogger;
Assert.ThatBool(
	actual := currentLogger <> initializationLogger,
	message := "An initialization setter must not assign a cyclic destination"
).IsTrue();
END_METHOD

(*!
<summary>Records manager behavior outside cyclic context without raising exceptions.</summary>
<description>
Uses persistent passive diagnostics and a dedicated ADS instance as an attempted assignment. The manager must
reject every logging call before filtering or counter changes, ignore assignment and do no cyclic work.
The cyclic test asserts these observations. The probe does not inject failures or allocate exceptions.
</description>
<param name="name">Name forwarded to the inherited test initializer for reporting.</param>
<param name="parent">Owning group forwarded to the inherited test initializer.</param>
*)
METHOD FB_init : BOOL
VAR_INPUT
	bInitRetains: BOOL; // TRUE: the retain variables are initialized (reset warm / reset cold)
	bInCopyCode: BOOL; // TRUE: the instance will be copied to the copy code afterward (online change)
	name : WSTRING;
	parent : TOF_Testing.ITestElement;
END_VAR
VAR
	taskIndex : DINT;
	loggerBefore : TOF_Core.ILogger;
	loggerAfter : TOF_Core.ILogger;
	totalBefore : ULINT;
	passedBefore : ULINT;
	message : TOF_Core.ERROR_MESSAGE := "non-cyclic initialization probe";
	messageAccepted : BOOL;
	errorAccepted : BOOL;
	exceptionAccepted : BOOL;
END_VAR
FB_init := TRUE;
taskIndex := TOF_Core.System.GetCurrentTaskIndex();

IF taskIndex >= 1 AND_THEN taskIndex <= TOF_Core.System.TASK_COUNT THEN
	RETURN;
END_IF

_InitializationContextObserved := TRUE;
loggerBefore := TOF_Core.LogManager.CurrentTaskLogger;
TOF_Core.LogManager.CurrentTaskLogger := _InitializationLogger;
loggerAfter := TOF_Core.LogManager.CurrentTaskLogger;
totalBefore := TOF_Core.LogManager.TotalMessageCounter;
passedBefore := TOF_Core.LogManager.PassedFilterMessageCounter;
messageAccepted := TOF_Core.LogManager.TryLogMessage(
	message := message,
	category := TOF_Core.LOG_CATEGORY.INFORMATION
);
errorAccepted := TOF_Core.LogManager.TryLogError(error := _InitializationError);
exceptionAccepted := TOF_Core.LogManager.TryLogException(
	exception := _InitializationException,
	severity := TOF_Core.ERROR_SEVERITY.ERROR
);
TOF_Core.LogManager.ExecuteCurrentTaskLogger();
_InitializationCallsRejected := loggerBefore = 0
	AND_THEN loggerAfter = 0
	AND_THEN NOT messageAccepted
	AND_THEN NOT errorAccepted
	AND_THEN NOT exceptionAccepted
	AND_THEN TOF_Core.LogManager.TotalMessageCounter = totalBefore
	AND_THEN TOF_Core.LogManager.PassedFilterMessageCounter = passedBefore;
END_METHOD

